(* IEC 61131-3 sources: smart-home/SmartHome/plc, 47 files *)

(* ---- Crosstable.gvl ---- *)
VAR_GLOBAL
	PLC_Iam_EP AT %QX0.4.0:BOOL;
	PLC_Iam_T1 AT %QX0.8.0:BOOL;
	PLC_Iam_T2 AT %QX0.12.0:BOOL;
	PLC_Iam_T3 AT %QX0.16.0:BOOL;
	PLC_Iam_T4 AT %QX0.20.0:BOOL;
	PLC_Iam_T5 AT %QX0.24.0:BOOL;
	PLC_Iam_T6 AT %QX0.28.0:BOOL;
	PLC_Iam_BA AT %QX0.32.0:BOOL;
	PLC_EP_exists AT %QX0.36.0:BOOL;
	PLC_Tn_count AT %QW0.40:UINT;	(* 0..6 *)
	PLC_BA_exists AT %QX0.44.0:BOOL;
	PLC_sunrise AT %QW0.48:UINT;	(* hh * 100 + mm *)
	PLC_sunset AT %QW0.52:UINT;	(* hh * 100 + mm *)
	PLC_day_brightness AT %QW0.56:UINT;
	PLC_night_brightness AT %QW0.60:UINT;
	PLC_screensaver AT %QW0.64:UINT;
	PLC_control_type AT %QW0.68:UINT;
	PLC_ConfigPassword AT %QD0.72:DINT;
	PLC_EP_enabled_wattmeters AT %QW0.80:UINT;	(* 0 .. 12 *)
	PLC_EP_enabled_relays AT %QW0.84:INT;	(* 0 .. 8 *)
	PLC_EP_overload_W AT %QW0.88:UINT;
	PLC_EP_max_assigned_W AT %QW0.92:UINT;
	PLC_EP_wattmeter_M_kWh_offset AT %QD0.96:DINT;	(* xxxxxxxxx.x kWh *)
	PLC_EP_wattmeter_M_e_kWh_offset AT %QD0.100:DINT;	(* xxxxxxxxx.x kWh *)
	PLC_EP_wattmeter_F_kWh_offset AT %QD0.104:DINT;	(* xxxxxxxxx.x kWh *)
	PLC_EP_wattmeter_F_e_kWh_offset AT %QD0.108:DINT;	(* xxxxxxxxx.x kWh *)
	PLC_EP_wattmeter01_kWh_offset AT %QD0.112:DINT;	(* xxxxxxxxx.x kWh *)
	PLC_EP_wattmeter02_kWh_offset AT %QD0.116:DINT;	(* xxxxxxxxx.x kWh *)
	PLC_EP_wattmeter03_kWh_offset AT %QD0.120:DINT;	(* xxxxxxxxx.x kWh *)
	PLC_EP_wattmeter04_kWh_offset AT %QD0.124:DINT;	(* xxxxxxxxx.x kWh *)
	PLC_EP_wattmeter05_kWh_offset AT %QD0.128:DINT;	(* xxxxxxxxx.x kWh *)
	PLC_EP_wattmeter06_kWh_offset AT %QD0.132:DINT;	(* xxxxxxxxx.x kWh *)
	PLC_EP_wattmeter07_kWh_offset AT %QD0.136:DINT;	(* xxxxxxxxx.x kWh *)
	PLC_EP_wattmeter08_kWh_offset AT %QD0.140:DINT;	(* xxxxxxxxx.x kWh *)
	PLC_EP_wattmeter09_kWh_offset AT %QD0.144:DINT;	(* xxxxxxxxx.x kWh *)
	PLC_EP_wattmeter10_kWh_offset AT %QD0.148:DINT;	(* xxxxxxxxx.x kWh *)
	PLC_T1_enabled_sensors AT %QW0.160:INT;
	PLC_T1_enabled_lamps AT %QW0.164:UINT;
	PLC_T1_max_request_W AT %QW0.168:UINT;
	PLC_T1_temperature_setpoint AT %QW0.172:INT;
	PLC_T1_humidity_setpoint AT %QW0.176:INT;
	PLC_T1_heating_status AT %QW0.180:INT;
	PLC_T1_temperature_setpoint_nt AT %QW0.184:INT;
	PLC_T1_humidity_setpoint_nt AT %QW0.188:INT;
	PLC_T1_daily_heating_s AT %QD0.192:UDINT;
	PLC_T1_monthly_heating_s AT %QD0.196:UDINT;
	PLC_T2_enabled_sensors AT %QW0.200:INT;
	PLC_T2_enabled_lamps AT %QW0.204:UINT;
	PLC_T2_max_request_W AT %QW0.208:UINT;
	PLC_T2_temperature_setpoint AT %QW0.212:INT;
	PLC_T2_humidity_setpoint AT %QW0.216:INT;
	PLC_T2_heating_status AT %QW0.220:INT;
	PLC_T2_temperature_setpoint_nt AT %QW0.224:INT;
	PLC_T2_humidity_setpoint_nt AT %QW0.228:INT;
	PLC_T2_daily_heating_s AT %QD0.232:UDINT;
	PLC_T2_monthly_heating_s AT %QD0.236:UDINT;
	PLC_T3_enabled_sensors AT %QW0.240:INT;
	PLC_T3_enabled_lamps AT %QW0.244:UINT;
	PLC_T3_max_request_W AT %QW0.248:UINT;
	PLC_T3_temperature_setpoint AT %QW0.252:INT;
	PLC_T3_humidity_setpoint AT %QW0.256:INT;
	PLC_T3_heating_status AT %QW0.260:INT;
	PLC_T3_temperature_setpoint_nt AT %QW0.264:INT;
	PLC_T3_humidity_setpoint_nt AT %QW0.268:INT;
	PLC_T3_daily_heating_s AT %QD0.272:UDINT;
	PLC_T3_monthly_heating_s AT %QD0.276:UDINT;
	PLC_T4_enabled_sensors AT %QW0.280:INT;
	PLC_T4_enabled_lamps AT %QW0.284:UINT;
	PLC_T4_max_request_W AT %QW0.288:UINT;
	PLC_T4_temperature_setpoint AT %QW0.292:INT;
	PLC_T4_humidity_setpoint AT %QW0.296:INT;
	PLC_T4_heating_status AT %QW0.300:INT;
	PLC_T4_temperature_setpoint_nt AT %QW0.304:INT;
	PLC_T4_humidity_setpoint_nt AT %QW0.308:INT;
	PLC_T4_daily_heating_s AT %QD0.312:UDINT;
	PLC_T4_monthly_heating_s AT %QD0.316:UDINT;
	PLC_T5_enabled_sensors AT %QW0.320:INT;
	PLC_T5_enabled_lamps AT %QW0.324:UINT;
	PLC_T5_max_request_W AT %QW0.328:UINT;
	PLC_T5_temperature_setpoint AT %QW0.332:INT;
	PLC_T5_humidity_setpoint AT %QW0.336:INT;
	PLC_T5_heating_status AT %QW0.340:INT;
	PLC_T5_temperature_setpoint_nt AT %QW0.344:INT;
	PLC_T5_humidity_setpoint_nt AT %QW0.348:INT;
	PLC_T5_daily_heating_s AT %QD0.352:UDINT;
	PLC_T5_monthly_heating_s AT %QD0.356:UDINT;
	PLC_T6_enabled_sensors AT %QW0.360:INT;
	PLC_T6_enabled_lamps AT %QW0.364:UINT;
	PLC_T6_max_request_W AT %QW0.368:UINT;
	PLC_T6_temperature_setpoint AT %QW0.372:INT;
	PLC_T6_humidity_setpoint AT %QW0.376:INT;
	PLC_T6_heating_status AT %QW0.380:INT;
	PLC_T6_temperature_setpoint_nt AT %QW0.384:INT;
	PLC_T6_humidity_setpoint_nt AT %QW0.388:INT;
	PLC_T6_daily_heating_s AT %QD0.392:UDINT;
	PLC_T6_monthly_heating_s AT %QD0.396:UDINT;
	PLC_BA_enabled_sensors AT %QW0.400:UINT;	(* 0, 8, 16, 24, 32 *)
	PLC_BA_daytime_bitmask AT %QD0.404:UDINT;
	PLC_BA_nighttime_bitmask AT %QD0.408:UDINT;
	PLC_BA_everything_bitmask AT %QD0.412:UDINT;
	PLC_BA_status AT %QW0.416:UINT;	(* ZERO, OFF, ARMED, ENABLED, RINGING, MUTED, TESTING *)
	PLC_BA_config_index AT %QW0.420:UINT;	(* 0 1 2 3 *)
	PLC_BA_password AT %QD0.424:DINT;
	Tsoglia_Resistenze AT %QW0.740:INT;	(* massima temperatura resistenze (50 .. 135 C) *)
	Tsoglia_Massetto AT %QW0.744:INT;	(* massima temperatura massetto (20 .. 30 C) *)
	Tsoglia_Ventola AT %QW0.748:INT;	(* minima temperatura ventole (50 .. 125 C) *)
	Vbase_Ventola AT %QW0.752:UINT;	(* valore base comando ventola (1.00V ..) *)
	TimerValue_1 AT %QD0.760:DINT;
	TimerValue_2 AT %QD0.764:DINT;
	PLC_RELOAD_CONF AT %QX0.772.0:BOOL;
	PLC_BA_just_started AT %QX0.776.0:BOOL;	(* just after init *)
	PLC_view_passwords AT %QX0.780.0:BOOL;
	PLC_buzzer_timer_1 AT %QX0.784.0:BOOL;
	PLC_buzzer_timer_2 AT %QX0.788.0:BOOL;
	PLC_buzzer_alarm AT %QX0.792.0:BOOL;
	PLC_buzzer_blackout_or_overload AT %QX0.796.0:BOOL;
	PLC_BA_ringing_flag AT %QX0.800.0:BOOL;
	PLC_BA_blackout_digin AT %QX0.804.0:BOOL;	(* Blackout detected flag *)
	PLC_EP_blackout_flag AT %QX0.808.0:BOOL;	(* Blackout detected flag *)
	PLC_EP_overload_flag AT %QX0.812.0:BOOL;	(* Overload detected flag *)
	PLC_EP_isOK AT %QX0.816.0:BOOL;
	PLC_T1_isOK AT %QX0.820.0:BOOL;
	PLC_T2_isOK AT %QX0.824.0:BOOL;
	PLC_T3_isOK AT %QX0.828.0:BOOL;
	PLC_T4_isOK AT %QX0.832.0:BOOL;
	PLC_T5_isOK AT %QX0.836.0:BOOL;
	PLC_T6_isOK AT %QX0.840.0:BOOL;
	PLC_BA_isOK AT %QX0.868.0:BOOL;
	PLC_BA_AlarmRinging AT %IX0.872.0:BOOL;	(* BA Alarm is ringing *)
	PLC_BA_BlackoutDetected AT %IX0.876.0:BOOL;	(* BA Blackout detected *)
	PLC_EP_BlackoutDetected AT %IX0.880.0:BOOL;	(* EP Blackout detected *)
	PLC_EP_OverloadDetected AT %IX0.884.0:BOOL;	(* EP Overload detected *)
	PLC_nighttime AT %QX0.888.0:BOOL;
	PLC_Tn_heating AT %QX0.892.0:BOOL;	(* al least one Tn is heating *)
	PLC_time_bis AT %QD0.912:REAL;	(* PLC_time + PLC_timeOffset *)
	PLC_timeMin_bis AT %QD0.916:REAL;	(* PLC_timeMin + PLC_timeOffset *)
	PLC_timeMax_bis AT %QD0.920:REAL;	(* PLC_timeMax + PLC_timeOffset *)
	PLC_timeOffset AT %QD0.924:REAL;	(* Graph display window *)
	TCP_EP_heartbeat AT %IW0.4000:UINT;	(* TCPS_STATUS NODE_09_STATUS *)
	TCP_EP_enabled_wattmeters AT %IW0.4004:UINT;	(* 0 .. 12 *)
	TCP_EP_wattmeters_ok AT %IW0.4008:UINT;	(* bit mask (node status) *)
	TCP_EP_wattmeter_M_W AT %IW0.4012:INT;	(* +/- xxxx W *)
	TCP_EP_wattmeter_M_var AT %IW0.4016:INT;	(* +/- xxxx var *)
	TCP_EP_wattmeter_M_VA AT %IW0.4020:INT;	(* +/- xxxx VA *)
	TCP_EP_wattmeter_M_pf AT %IW0.4024:INT;	(* +/- x.xxx *)
	TCP_EP_wattmeter_M_Hz AT %IW0.4028:INT;	(* xxx.xx Hz *)
	TCP_EP_wattmeter_M_V AT %IW0.4032:INT;	(* xxx.xx V *)
	TCP_EP_wattmeter_M_A AT %IW0.4036:INT;	(* xx.xxx A *)
	TCP_EP_wattmeter_M_kWh AT %ID0.4040:DINT;	(* xxxxxxxxx.x +kWh *)
	TCP_EP_wattmeter_M_e_kWh AT %ID0.4044:DINT;	(* xxxxxxxxx.x -kWh *)
	TCP_EP_wattmeter_F_W AT %IW0.4048:INT;	(* +/- xxxx W *)
	TCP_EP_wattmeter_F_var AT %IW0.4052:INT;	(* +/- xxxx var *)
	TCP_EP_wattmeter_F_VA AT %IW0.4056:INT;	(* +/- xxxx VA *)
	TCP_EP_wattmeter_F_pf AT %IW0.4060:INT;	(* +/- x.xxx *)
	TCP_EP_wattmeter_F_Hz AT %IW0.4064:INT;	(* xxx.xx Hz *)
	TCP_EP_wattmeter_F_V AT %IW0.4068:INT;	(* xxx.xx V *)
	TCP_EP_wattmeter_F_A AT %IW0.4072:INT;	(* xx.xxx A *)
	TCP_EP_wattmeter_F_kWh AT %ID0.4076:DINT;	(* xxxxxxxxx.x +kWh *)
	TCP_EP_wattmeter_F_e_kWh AT %ID0.4080:DINT;	(* xxxxxxxxx.x -kWh *)
	TCP_EP_wattmeter01_W AT %IW0.4084:INT;	(* +/- xxxx W *)
	TCP_EP_wattmeter01_var AT %IW0.4088:INT;	(* +/- xxxx var *)
	TCP_EP_wattmeter01_VA AT %IW0.4092:INT;	(* +/- xxxx VA *)
	TCP_EP_wattmeter01_kWh AT %ID0.4096:DINT;	(* xxxxxxxxx.x +kWh *)
	TCP_EP_wattmeter02_W AT %IW0.4100:INT;	(* +/- xxxx W *)
	TCP_EP_wattmeter02_var AT %IW0.4104:INT;	(* +/- xxxx var *)
	TCP_EP_wattmeter02_VA AT %IW0.4108:INT;	(* +/- xxxx VA *)
	TCP_EP_wattmeter02_kWh AT %ID0.4112:DINT;	(* xxxxxxxxx.x +kWh *)
	TCP_EP_wattmeter03_W AT %IW0.4116:INT;	(* +/- xxxx W *)
	TCP_EP_wattmeter03_var AT %IW0.4120:INT;	(* +/- xxxx var *)
	TCP_EP_wattmeter03_VA AT %IW0.4124:INT;	(* +/- xxxx VA *)
	TCP_EP_wattmeter03_kWh AT %ID0.4128:DINT;	(* xxxxxxxxx.x +kWh *)
	TCP_EP_wattmeter04_W AT %IW0.4132:INT;	(* +/- xxxx W *)
	TCP_EP_wattmeter04_var AT %IW0.4136:INT;	(* +/- xxxx var *)
	TCP_EP_wattmeter04_VA AT %IW0.4140:INT;	(* +/- xxxx VA *)
	TCP_EP_wattmeter04_kWh AT %ID0.4144:DINT;	(* xxxxxxxxx.x +kWh *)
	TCP_EP_wattmeter05_W AT %IW0.4148:INT;	(* +/- xxxx W *)
	TCP_EP_wattmeter05_var AT %IW0.4152:INT;	(* +/- xxxx var *)
	TCP_EP_wattmeter05_VA AT %IW0.4156:INT;	(* +/- xxxx VA *)
	TCP_EP_wattmeter05_kWh AT %ID0.4160:DINT;	(* xxxxxxxxx.x +kWh *)
	TCP_EP_wattmeter06_W AT %IW0.4164:INT;	(* +/- xxxx W *)
	TCP_EP_wattmeter06_var AT %IW0.4168:INT;	(* +/- xxxx var *)
	TCP_EP_wattmeter06_VA AT %IW0.4172:INT;	(* +/- xxxx VA *)
	TCP_EP_wattmeter06_kWh AT %ID0.4176:DINT;	(* xxxxxxxxx.x +kWh *)
	TCP_EP_wattmeter07_W AT %IW0.4180:INT;	(* +/- xxxx W *)
	TCP_EP_wattmeter07_var AT %IW0.4184:INT;	(* +/- xxxx var *)
	TCP_EP_wattmeter07_VA AT %IW0.4188:INT;	(* +/- xxxx VA *)
	TCP_EP_wattmeter07_kWh AT %ID0.4192:DINT;	(* xxxxxxxxx.x +kWh *)
	TCP_EP_wattmeter08_W AT %IW0.4196:INT;	(* +/- xxxx W *)
	TCP_EP_wattmeter08_var AT %IW0.4200:INT;	(* +/- xxxx var *)
	TCP_EP_wattmeter08_VA AT %IW0.4204:INT;	(* +/- xxxx VA *)
	TCP_EP_wattmeter08_kWh AT %ID0.4208:DINT;	(* xxxxxxxxx.x +kWh *)
	TCP_EP_wattmeter09_W AT %IW0.4212:INT;	(* +/- xxxx W *)
	TCP_EP_wattmeter09_var AT %IW0.4216:INT;	(* +/- xxxx var *)
	TCP_EP_wattmeter09_VA AT %IW0.4220:INT;	(* +/- xxxx VA *)
	TCP_EP_wattmeter09_kWh AT %ID0.4224:DINT;	(* xxxxxxxxx.x +kWh *)
	TCP_EP_wattmeter10_W AT %IW0.4228:INT;	(* +/- xxxx W *)
	TCP_EP_wattmeter10_var AT %IW0.4232:INT;	(* +/- xxxx var *)
	TCP_EP_wattmeter10_VA AT %IW0.4236:INT;	(* +/- xxxx VA *)
	TCP_EP_wattmeter10_kWh AT %ID0.4240:DINT;	(* xxxxxxxxx.x +kWh *)
	TCP_EP_BlackoutDetected AT %IX0.4244.0:BOOL;
	TCP_EP_OverloadDetected AT %IX0.4248.0:BOOL;
	TCP_EP_enabled_relays AT %IW0.4252:INT;	(* 0 .. 8 *)
	TCP_EP_relay_A AT %QX0.4256.0:BOOL;
	TCP_EP_relay_B AT %QX0.4260.0:BOOL;
	TCP_EP_relay_C AT %QX0.4264.0:BOOL;
	TCP_EP_relay_D AT %QX0.4268.0:BOOL;
	TCP_EP_relay_E AT %QX0.4272.0:BOOL;
	TCP_EP_relay_F AT %QX0.4276.0:BOOL;
	TCP_EP_relay_G AT %QX0.4280.0:BOOL;
	TCP_EP_relay_H AT %QX0.4284.0:BOOL;
	TCP_EP_overload_W AT %IW0.4288:UINT;
	TCP_EP_max_assigned_W AT %IW0.4292:UINT;
	TCP_EP_tic_in_tac AT %IW0.4296:UINT;
	TCP_EP_requested_W AT %IW0.4300:UINT;
	TCP_EP_T1_assigned_W AT %IW0.4304:UINT;
	TCP_EP_T2_assigned_W AT %IW0.4308:UINT;
	TCP_EP_T3_assigned_W AT %IW0.4312:UINT;
	TCP_EP_T4_assigned_W AT %IW0.4316:UINT;
	TCP_EP_T5_assigned_W AT %IW0.4320:UINT;
	TCP_EP_T6_assigned_W AT %IW0.4324:UINT;
	TCP_EP_assigned_W AT %IW0.4328:UINT;
	TCP_EP_control_type AT %IW0.4332:UINT;
	TCP_T1_heartbeat AT %IW0.4400:UINT;	(* TCP1_STATUS NODE_02_STATUS *)
	TCP_T1_enabled_sensors AT %IW0.4404:INT;
	TCP_T1_temperature AT %IW0.4408:INT;
	TCP_T1_temperature_bis AT %IW0.4412:INT;
	TCP_T1_temperature_ext AT %IW0.4416:INT;
	TCP_T1_humidity AT %IW0.4420:INT;
	TCP_T1_humidity_bis AT %IW0.4424:INT;
	TCP_T1_humidity_ext AT %IW0.4428:INT;
	TCP_T1_temperature_setpoint AT %QW0.4432:INT;
	TCP_T1_humidity_setpoint AT %QW0.4436:INT;
	TCP_T1_enabled_lamps AT %IW0.4440:UINT;
	TCP_T1_lamp_1 AT %QX0.4444.0:BOOL;
	TCP_T1_lamp_2 AT %QX0.4448.0:BOOL;
	TCP_T1_lamp_3 AT %QX0.4452.0:BOOL;
	TCP_T1_lamp_4 AT %QX0.4456.0:BOOL;
	TCP_T1_lamp_5 AT %QX0.4460.0:BOOL;
	TCP_T1_max_request_W AT %IW0.4464:UINT;
	TCP_T1_heating AT %IX0.4468.0:BOOL;
	TCP_T1_nighttime AT %IX0.4472.0:BOOL;
	TCP_T1_heating_status AT %QW0.4476:INT;
	TCP_T1_heating_timer AT %QW0.4480:INT;	(* seconds (max 9 h) *)
	TCP_T1_sunrise AT %QW0.4484:UINT;	(* hh * 100 + mm *)
	TCP_T1_sunset AT %QW0.4488:UINT;	(* hh * 100 + mm *)
	TCP_T1_temperature_setpoint_nt AT %QW0.4492:INT;
	TCP_T1_humidity_setpoint_nt AT %QW0.4496:INT;
	TCP_T1_lamp_feedback_1 AT %IX0.4500.0:BOOL;
	TCP_T1_lamp_feedback_2 AT %IX0.4504.0:BOOL;
	TCP_T1_lamp_feedback_3 AT %IX0.4508.0:BOOL;
	TCP_T1_lamp_feedback_4 AT %IX0.4512.0:BOOL;
	TCP_T1_lamp_feedback_5 AT %IX0.4516.0:BOOL;
	TCP_T1_requested_W AT %IW0.4520:UINT;
	TCP_T1_control_type AT %IW0.4524:UINT;
	TCP_T1_daily_heating_s AT %ID0.4528:UDINT;
	TCP_T1_monthly_heating_s AT %ID0.4532:UDINT;
	TCP_T2_heartbeat AT %IW0.4600:UINT;	(* TCP2_STATUS NODE_03_STATUS *)
	TCP_T2_enabled_sensors AT %IW0.4604:INT;
	TCP_T2_temperature AT %IW0.4608:INT;
	TCP_T2_temperature_bis AT %IW0.4612:INT;
	TCP_T2_temperature_ext AT %IW0.4616:INT;
	TCP_T2_humidity AT %IW0.4620:INT;
	TCP_T2_humidity_bis AT %IW0.4624:INT;
	TCP_T2_humidity_ext AT %IW0.4628:INT;
	TCP_T2_temperature_setpoint AT %QW0.4632:INT;
	TCP_T2_humidity_setpoint AT %QW0.4636:INT;
	TCP_T2_enabled_lamps AT %IW0.4640:UINT;
	TCP_T2_lamp_1 AT %QX0.4644.0:BOOL;
	TCP_T2_lamp_2 AT %QX0.4648.0:BOOL;
	TCP_T2_lamp_3 AT %QX0.4652.0:BOOL;
	TCP_T2_lamp_4 AT %QX0.4656.0:BOOL;
	TCP_T2_lamp_5 AT %QX0.4660.0:BOOL;
	TCP_T2_max_request_W AT %IW0.4664:UINT;
	TCP_T2_heating AT %IX0.4668.0:BOOL;
	TCP_T2_nighttime AT %IX0.4672.0:BOOL;
	TCP_T2_heating_status AT %QW0.4676:INT;
	TCP_T2_heating_timer AT %QW0.4680:INT;	(* seconds (max 9 h) *)
	TCP_T2_sunrise AT %QW0.4684:UINT;	(* hh * 100 + mm *)
	TCP_T2_sunset AT %QW0.4688:UINT;	(* hh * 100 + mm *)
	TCP_T2_temperature_setpoint_nt AT %QW0.4692:INT;
	TCP_T2_humidity_setpoint_nt AT %QW0.4696:INT;
	TCP_T2_lamp_feedback_1 AT %IX0.4700.0:BOOL;
	TCP_T2_lamp_feedback_2 AT %IX0.4704.0:BOOL;
	TCP_T2_lamp_feedback_3 AT %IX0.4708.0:BOOL;
	TCP_T2_lamp_feedback_4 AT %IX0.4712.0:BOOL;
	TCP_T2_lamp_feedback_5 AT %IX0.4716.0:BOOL;
	TCP_T2_requested_W AT %IW0.4720:UINT;
	TCP_T2_control_type AT %IW0.4724:UINT;
	TCP_T2_daily_heating_s AT %ID0.4728:UDINT;
	TCP_T2_monthly_heating_s AT %ID0.4732:UDINT;
	TCP_T3_heartbeat AT %IW0.4800:UINT;	(* TCP3_STATUS NODE_04_STATUS *)
	TCP_T3_enabled_sensors AT %IW0.4804:INT;
	TCP_T3_temperature AT %IW0.4808:INT;
	TCP_T3_temperature_bis AT %IW0.4812:INT;
	TCP_T3_temperature_ext AT %IW0.4816:INT;
	TCP_T3_humidity AT %IW0.4820:INT;
	TCP_T3_humidity_bis AT %IW0.4824:INT;
	TCP_T3_humidity_ext AT %IW0.4828:INT;
	TCP_T3_temperature_setpoint AT %QW0.4832:INT;
	TCP_T3_humidity_setpoint AT %QW0.4836:INT;
	TCP_T3_enabled_lamps AT %IW0.4840:UINT;
	TCP_T3_lamp_1 AT %QX0.4844.0:BOOL;
	TCP_T3_lamp_2 AT %QX0.4848.0:BOOL;
	TCP_T3_lamp_3 AT %QX0.4852.0:BOOL;
	TCP_T3_lamp_4 AT %QX0.4856.0:BOOL;
	TCP_T3_lamp_5 AT %QX0.4860.0:BOOL;
	TCP_T3_max_request_W AT %IW0.4864:UINT;
	TCP_T3_heating AT %IX0.4868.0:BOOL;
	TCP_T3_nighttime AT %IX0.4872.0:BOOL;
	TCP_T3_heating_status AT %QW0.4876:INT;
	TCP_T3_heating_timer AT %QW0.4880:INT;	(* seconds (max 9 h) *)
	TCP_T3_sunrise AT %QW0.4884:UINT;	(* hh * 100 + mm *)
	TCP_T3_sunset AT %QW0.4888:UINT;	(* hh * 100 + mm *)
	TCP_T3_temperature_setpoint_nt AT %QW0.4892:INT;
	TCP_T3_humidity_setpoint_nt AT %QW0.4896:INT;
	TCP_T3_lamp_feedback_1 AT %IX0.4900.0:BOOL;
	TCP_T3_lamp_feedback_2 AT %IX0.4904.0:BOOL;
	TCP_T3_lamp_feedback_3 AT %IX0.4908.0:BOOL;
	TCP_T3_lamp_feedback_4 AT %IX0.4912.0:BOOL;
	TCP_T3_lamp_feedback_5 AT %IX0.4916.0:BOOL;
	TCP_T3_requested_W AT %IW0.4920:UINT;
	TCP_T3_control_type AT %IW0.4924:UINT;
	TCP_T3_daily_heating_s AT %ID0.4928:UDINT;
	TCP_T3_monthly_heating_s AT %ID0.4932:UDINT;
	TCP_T4_heartbeat AT %IW0.5000:UINT;	(* TCP4_STATUS NODE_05_STATUS *)
	TCP_T4_enabled_sensors AT %IW0.5004:INT;
	TCP_T4_temperature AT %IW0.5008:INT;
	TCP_T4_temperature_bis AT %IW0.5012:INT;
	TCP_T4_temperature_ext AT %IW0.5016:INT;
	TCP_T4_humidity AT %IW0.5020:INT;
	TCP_T4_humidity_bis AT %IW0.5024:INT;
	TCP_T4_humidity_ext AT %IW0.5028:INT;
	TCP_T4_temperature_setpoint AT %QW0.5032:INT;
	TCP_T4_humidity_setpoint AT %QW0.5036:INT;
	TCP_T4_enabled_lamps AT %IW0.5040:UINT;
	TCP_T4_lamp_1 AT %QX0.5044.0:BOOL;
	TCP_T4_lamp_2 AT %QX0.5048.0:BOOL;
	TCP_T4_lamp_3 AT %QX0.5052.0:BOOL;
	TCP_T4_lamp_4 AT %QX0.5056.0:BOOL;
	TCP_T4_lamp_5 AT %QX0.5060.0:BOOL;
	TCP_T4_max_request_W AT %IW0.5064:UINT;
	TCP_T4_heating AT %IX0.5068.0:BOOL;
	TCP_T4_nighttime AT %IX0.5072.0:BOOL;
	TCP_T4_heating_status AT %QW0.5076:INT;
	TCP_T4_heating_timer AT %QW0.5080:INT;	(* seconds (max 9 h) *)
	TCP_T4_sunrise AT %QW0.5084:UINT;	(* hh * 100 + mm *)
	TCP_T4_sunset AT %QW0.5088:UINT;	(* hh * 100 + mm *)
	TCP_T4_temperature_setpoint_nt AT %QW0.5092:INT;
	TCP_T4_humidity_setpoint_nt AT %QW0.5096:INT;
	TCP_T4_lamp_feedback_1 AT %IX0.5100.0:BOOL;
	TCP_T4_lamp_feedback_2 AT %IX0.5104.0:BOOL;
	TCP_T4_lamp_feedback_3 AT %IX0.5108.0:BOOL;
	TCP_T4_lamp_feedback_4 AT %IX0.5112.0:BOOL;
	TCP_T4_lamp_feedback_5 AT %IX0.5116.0:BOOL;
	TCP_T4_requested_W AT %IW0.5120:UINT;
	TCP_T4_control_type AT %IW0.5124:UINT;
	TCP_T4_daily_heating_s AT %ID0.5128:UDINT;
	TCP_T4_monthly_heating_s AT %ID0.5132:UDINT;
	TCP_T5_heartbeat AT %IW0.5200:UINT;	(* TCP5_STATUS NODE_06_STATUS *)
	TCP_T5_enabled_sensors AT %IW0.5204:INT;
	TCP_T5_temperature AT %IW0.5208:INT;
	TCP_T5_temperature_bis AT %IW0.5212:INT;
	TCP_T5_temperature_ext AT %IW0.5216:INT;
	TCP_T5_humidity AT %IW0.5220:INT;
	TCP_T5_humidity_bis AT %IW0.5224:INT;
	TCP_T5_humidity_ext AT %IW0.5228:INT;
	TCP_T5_temperature_setpoint AT %QW0.5232:INT;
	TCP_T5_humidity_setpoint AT %QW0.5236:INT;
	TCP_T5_enabled_lamps AT %IW0.5240:UINT;
	TCP_T5_lamp_1 AT %QX0.5244.0:BOOL;
	TCP_T5_lamp_2 AT %QX0.5248.0:BOOL;
	TCP_T5_lamp_3 AT %QX0.5252.0:BOOL;
	TCP_T5_lamp_4 AT %QX0.5256.0:BOOL;
	TCP_T5_lamp_5 AT %QX0.5260.0:BOOL;
	TCP_T5_max_request_W AT %IW0.5264:UINT;
	TCP_T5_heating AT %IX0.5268.0:BOOL;
	TCP_T5_nighttime AT %IX0.5272.0:BOOL;
	TCP_T5_heating_status AT %QW0.5276:INT;
	TCP_T5_heating_timer AT %QW0.5280:INT;	(* seconds (max 9 h) *)
	TCP_T5_sunrise AT %QW0.5284:UINT;	(* hh * 100 + mm *)
	TCP_T5_sunset AT %QW0.5288:UINT;	(* hh * 100 + mm *)
	TCP_T5_temperature_setpoint_nt AT %QW0.5292:INT;
	TCP_T5_humidity_setpoint_nt AT %QW0.5296:INT;
	TCP_T5_lamp_feedback_1 AT %IX0.5300.0:BOOL;
	TCP_T5_lamp_feedback_2 AT %IX0.5304.0:BOOL;
	TCP_T5_lamp_feedback_3 AT %IX0.5308.0:BOOL;
	TCP_T5_lamp_feedback_4 AT %IX0.5312.0:BOOL;
	TCP_T5_lamp_feedback_5 AT %IX0.5316.0:BOOL;
	TCP_T5_requested_W AT %IW0.5320:UINT;
	TCP_T5_control_type AT %IW0.5324:UINT;
	TCP_T5_daily_heating_s AT %ID0.5328:UDINT;
	TCP_T5_monthly_heating_s AT %ID0.5332:UDINT;
	TCP_T6_heartbeat AT %IW0.5400:UINT;	(* TCP6_STATUS NODE_07_STATUS *)
	TCP_T6_enabled_sensors AT %IW0.5404:INT;
	TCP_T6_temperature AT %IW0.5408:INT;
	TCP_T6_temperature_bis AT %IW0.5412:INT;
	TCP_T6_temperature_ext AT %IW0.5416:INT;
	TCP_T6_humidity AT %IW0.5420:INT;
	TCP_T6_humidity_bis AT %IW0.5424:INT;
	TCP_T6_humidity_ext AT %IW0.5428:INT;
	TCP_T6_temperature_setpoint AT %QW0.5432:INT;
	TCP_T6_humidity_setpoint AT %QW0.5436:INT;
	TCP_T6_enabled_lamps AT %IW0.5440:UINT;
	TCP_T6_lamp_1 AT %QX0.5444.0:BOOL;
	TCP_T6_lamp_2 AT %QX0.5448.0:BOOL;
	TCP_T6_lamp_3 AT %QX0.5452.0:BOOL;
	TCP_T6_lamp_4 AT %QX0.5456.0:BOOL;
	TCP_T6_lamp_5 AT %QX0.5460.0:BOOL;
	TCP_T6_max_request_W AT %IW0.5464:UINT;
	TCP_T6_heating AT %IX0.5468.0:BOOL;
	TCP_T6_nighttime AT %IX0.5472.0:BOOL;
	TCP_T6_heating_status AT %QW0.5476:INT;
	TCP_T6_heating_timer AT %QW0.5480:INT;	(* seconds (max 9 h) *)
	TCP_T6_sunrise AT %QW0.5484:UINT;	(* hh * 100 + mm *)
	TCP_T6_sunset AT %QW0.5488:UINT;	(* hh * 100 + mm *)
	TCP_T6_temperature_setpoint_nt AT %QW0.5492:INT;
	TCP_T6_humidity_setpoint_nt AT %QW0.5496:INT;
	TCP_T6_lamp_feedback_1 AT %IX0.5500.0:BOOL;
	TCP_T6_lamp_feedback_2 AT %IX0.5504.0:BOOL;
	TCP_T6_lamp_feedback_3 AT %IX0.5508.0:BOOL;
	TCP_T6_lamp_feedback_4 AT %IX0.5512.0:BOOL;
	TCP_T6_lamp_feedback_5 AT %IX0.5516.0:BOOL;
	TCP_T6_requested_W AT %IW0.5520:UINT;
	TCP_T6_control_type AT %IW0.5524:UINT;
	TCP_T6_daily_heating_s AT %ID0.5528:UDINT;
	TCP_T6_monthly_heating_s AT %ID0.5532:UDINT;
	TCP_BA_heartbeat AT %IW0.6800:UINT;	(* TCP7_STATUS NODE_08_STATUS *)
	TCP_BA_enabled_sensors AT %IW0.6804:UINT;	(* 0, 8, 16, 24, 32 *)
	TCP_BA_status AT %IW0.6808:UINT;	(* ZERO, OFF, ARMED, ENABLED, RINGING, MUTED, TESTING *)
	TCP_BA_config_index AT %IW0.6812:UINT;	(* 0 1 2 3 *)
	TCP_BA_config_mask AT %ID0.6816:UDINT;	(* bit mask *)
	TCP_BA_led_green AT %IX0.6820.0:BOOL;	(* ARMED(blinking), ENABLED, RINGING, MUTED *)
	TCP_BA_led_red AT %IX0.6824.0:BOOL;	(* ARMED(if NG), RINGING(blinking), MUTED *)
	TCP_BA_led_yellow1 AT %IX0.6828.0:BOOL;	(* NIGHTIME, EVERYTHING *)
	TCP_BA_led_yellow2 AT %IX0.6832.0:BOOL;	(* DAYTIME, EVERYTHING *)
	TCP_BA_siren AT %IX0.6836.0:BOOL;	(* HPA *)
	TCP_BA_relay_A AT %IX0.6840.0:BOOL;
	TCP_BA_relay_B AT %IX0.6844.0:BOOL;
	TCP_BA_relay_C AT %IX0.6848.0:BOOL;
	TCP_BA_input_9 AT %IX0.6852.0:BOOL;
	TCP_BA_input_10 AT %IX0.6856.0:BOOL;
	TCP_BA_input_11 AT %IX0.6860.0:BOOL;
	TCP_BA_input_12 AT %IX0.6864.0:BOOL;
	TCP_BA_BlackoutDetected AT %IX0.6868.0:BOOL;
	TCP_BA_command AT %QD0.6872:UDINT;	(* NONE, ARM, NOTHING, DAYTIME, NIGHTIME, EVERYTHING, ENABLE, DISABLE, ACK, TEST *)
	TCP_BA_OK_1 AT %IW0.6876:UINT;
	TCP_BA_OK_2 AT %IW0.6880:UINT;
	TCP_BA_OK_3 AT %IW0.6884:UINT;
	TCP_BA_OK_4 AT %IW0.6888:UINT;
	TCP_BA_OK_5 AT %IW0.6892:UINT;
	TCP_BA_OK_6 AT %IW0.6896:UINT;
	TCP_BA_OK_7 AT %IW0.6900:UINT;
	TCP_BA_OK_8 AT %IW0.6904:UINT;
	TCP_BA_OK_9 AT %IW0.6908:UINT;
	TCP_BA_OK_10 AT %IW0.6912:UINT;
	TCP_BA_OK_11 AT %IW0.6916:UINT;
	TCP_BA_OK_12 AT %IW0.6920:UINT;
	TCP_BA_OK_13 AT %IW0.6924:UINT;
	TCP_BA_OK_14 AT %IW0.6928:UINT;
	TCP_BA_OK_15 AT %IW0.6932:UINT;
	TCP_BA_OK_16 AT %IW0.6936:UINT;
	TCP_BA_OK_17 AT %IW0.6940:UINT;
	TCP_BA_OK_18 AT %IW0.6944:UINT;
	TCP_BA_OK_19 AT %IW0.6948:UINT;
	TCP_BA_OK_20 AT %IW0.6952:UINT;
	TCP_BA_OK_21 AT %IW0.6956:UINT;
	TCP_BA_OK_22 AT %IW0.6960:UINT;
	TCP_BA_OK_23 AT %IW0.6964:UINT;
	TCP_BA_OK_24 AT %IW0.6968:UINT;
	TCP_BA_OK_25 AT %IW0.6972:UINT;
	TCP_BA_OK_26 AT %IW0.6976:UINT;
	TCP_BA_OK_27 AT %IW0.6980:UINT;
	TCP_BA_OK_28 AT %IW0.6984:UINT;
	TCP_BA_OK_29 AT %IW0.6988:UINT;
	TCP_BA_OK_30 AT %IW0.6992:UINT;
	TCP_BA_OK_31 AT %IW0.6996:UINT;
	TCP_BA_OK_32 AT %IW0.7000:UINT;
	TCP_BA_control_type AT %IW0.7004:UINT;
	SRV_EP_heartbeat AT %QW0.8000:UINT;	(* TCPS_STATUS NODE_09_STATUS *)
	SRV_EP_enabled_wattmeters AT %QW0.8004:UINT;	(* 0 .. 12 *)
	SRV_EP_wattmeters_ok AT %QW0.8008:UINT;	(* bit mask (node status) *)
	SRV_EP_wattmeter_M_W AT %QW0.8012:INT;	(* +/- xxxx W *)
	SRV_EP_wattmeter_M_var AT %QW0.8016:INT;	(* +/- xxxx var *)
	SRV_EP_wattmeter_M_VA AT %QW0.8020:INT;	(* +/- xxxx VA *)
	SRV_EP_wattmeter_M_pf AT %QW0.8024:INT;	(* +/- x.xxx *)
	SRV_EP_wattmeter_M_Hz AT %QW0.8028:INT;	(* xxx.xx Hz *)
	SRV_EP_wattmeter_M_V AT %QW0.8032:INT;	(* xxx.xx V *)
	SRV_EP_wattmeter_M_A AT %QW0.8036:INT;	(* xx.xxx A *)
	SRV_EP_wattmeter_M_kWh AT %QD0.8040:DINT;	(* xxxxxxxxx.x +kWh *)
	SRV_EP_wattmeter_M_e_kWh AT %QD0.8044:DINT;	(* xxxxxxxxx.x -kWh *)
	SRV_EP_wattmeter_F_W AT %QW0.8048:INT;	(* +/- xxxx W *)
	SRV_EP_wattmeter_F_var AT %QW0.8052:INT;	(* +/- xxxx var *)
	SRV_EP_wattmeter_F_VA AT %QW0.8056:INT;	(* +/- xxxx VA *)
	SRV_EP_wattmeter_F_pf AT %QW0.8060:INT;	(* +/- x.xxx *)
	SRV_EP_wattmeter_F_Hz AT %QW0.8064:INT;	(* xxx.xx Hz *)
	SRV_EP_wattmeter_F_V AT %QW0.8068:INT;	(* xxx.xx V *)
	SRV_EP_wattmeter_F_A AT %QW0.8072:INT;	(* xx.xxx A *)
	SRV_EP_wattmeter_F_kWh AT %QD0.8076:DINT;	(* xxxxxxxxx.x +kWh *)
	SRV_EP_wattmeter_F_e_kWh AT %QD0.8080:DINT;	(* xxxxxxxxx.x -kWh *)
	SRV_EP_wattmeter01_W AT %QW0.8084:INT;	(* +/- xxxx W *)
	SRV_EP_wattmeter01_var AT %QW0.8088:INT;	(* +/- xxxx var *)
	SRV_EP_wattmeter01_VA AT %QW0.8092:INT;	(* +/- xxxx VA *)
	SRV_EP_wattmeter01_kWh AT %QD0.8096:DINT;	(* xxxxxxxxx.x +kWh *)
	SRV_EP_wattmeter02_W AT %QW0.8100:INT;	(* +/- xxxx W *)
	SRV_EP_wattmeter02_var AT %QW0.8104:INT;	(* +/- xxxx var *)
	SRV_EP_wattmeter02_VA AT %QW0.8108:INT;	(* +/- xxxx VA *)
	SRV_EP_wattmeter02_kWh AT %QD0.8112:DINT;	(* xxxxxxxxx.x +kWh *)
	SRV_EP_wattmeter03_W AT %QW0.8116:INT;	(* +/- xxxx W *)
	SRV_EP_wattmeter03_var AT %QW0.8120:INT;	(* +/- xxxx var *)
	SRV_EP_wattmeter03_VA AT %QW0.8124:INT;	(* +/- xxxx VA *)
	SRV_EP_wattmeter03_kWh AT %QD0.8128:DINT;	(* xxxxxxxxx.x +kWh *)
	SRV_EP_wattmeter04_W AT %QW0.8132:INT;	(* +/- xxxx W *)
	SRV_EP_wattmeter04_var AT %QW0.8136:INT;	(* +/- xxxx var *)
	SRV_EP_wattmeter04_VA AT %QW0.8140:INT;	(* +/- xxxx VA *)
	SRV_EP_wattmeter04_kWh AT %QD0.8144:DINT;	(* xxxxxxxxx.x +kWh *)
	SRV_EP_wattmeter05_W AT %QW0.8148:INT;	(* +/- xxxx W *)
	SRV_EP_wattmeter05_var AT %QW0.8152:INT;	(* +/- xxxx var *)
	SRV_EP_wattmeter05_VA AT %QW0.8156:INT;	(* +/- xxxx VA *)
	SRV_EP_wattmeter05_kWh AT %QD0.8160:DINT;	(* xxxxxxxxx.x +kWh *)
	SRV_EP_wattmeter06_W AT %QW0.8164:INT;	(* +/- xxxx W *)
	SRV_EP_wattmeter06_var AT %QW0.8168:INT;	(* +/- xxxx var *)
	SRV_EP_wattmeter06_VA AT %QW0.8172:INT;	(* +/- xxxx VA *)
	SRV_EP_wattmeter06_kWh AT %QD0.8176:DINT;	(* xxxxxxxxx.x +kWh *)
	SRV_EP_wattmeter07_W AT %QW0.8180:INT;	(* +/- xxxx W *)
	SRV_EP_wattmeter07_var AT %QW0.8184:INT;	(* +/- xxxx var *)
	SRV_EP_wattmeter07_VA AT %QW0.8188:INT;	(* +/- xxxx VA *)
	SRV_EP_wattmeter07_kWh AT %QD0.8192:DINT;	(* xxxxxxxxx.x +kWh *)
	SRV_EP_wattmeter08_W AT %QW0.8196:INT;	(* +/- xxxx W *)
	SRV_EP_wattmeter08_var AT %QW0.8200:INT;	(* +/- xxxx var *)
	SRV_EP_wattmeter08_VA AT %QW0.8204:INT;	(* +/- xxxx VA *)
	SRV_EP_wattmeter08_kWh AT %QD0.8208:DINT;	(* xxxxxxxxx.x +kWh *)
	SRV_EP_wattmeter09_W AT %QW0.8212:INT;	(* +/- xxxx W *)
	SRV_EP_wattmeter09_var AT %QW0.8216:INT;	(* +/- xxxx var *)
	SRV_EP_wattmeter09_VA AT %QW0.8220:INT;	(* +/- xxxx VA *)
	SRV_EP_wattmeter09_kWh AT %QD0.8224:DINT;	(* xxxxxxxxx.x +kWh *)
	SRV_EP_wattmeter10_W AT %QW0.8228:INT;	(* +/- xxxx W *)
	SRV_EP_wattmeter10_var AT %QW0.8232:INT;	(* +/- xxxx var *)
	SRV_EP_wattmeter10_VA AT %QW0.8236:INT;	(* +/- xxxx VA *)
	SRV_EP_wattmeter10_kWh AT %QD0.8240:DINT;	(* xxxxxxxxx.x +kWh *)
	SRV_EP_BlackoutDetected AT %QX0.8244.0:BOOL;
	SRV_EP_OverloadDetected AT %QX0.8248.0:BOOL;
	SRV_EP_enabled_relays AT %QW0.8252:INT;	(* 0 .. 8 *)
	SRV_EP_relay_A AT %QX0.8256.0:BOOL;
	SRV_EP_relay_B AT %QX0.8260.0:BOOL;
	SRV_EP_relay_C AT %QX0.8264.0:BOOL;
	SRV_EP_relay_D AT %QX0.8268.0:BOOL;
	SRV_EP_relay_E AT %QX0.8272.0:BOOL;
	SRV_EP_relay_F AT %QX0.8276.0:BOOL;
	SRV_EP_relay_G AT %QX0.8280.0:BOOL;
	SRV_EP_relay_H AT %QX0.8284.0:BOOL;
	SRV_EP_overload_W AT %QW0.8288:UINT;
	SRV_EP_max_assigned_W AT %QW0.8292:UINT;
	SRV_EP_tic_in_tac AT %QW0.8296:UINT;
	SRV_EP_requested_W AT %QW0.8300:UINT;
	SRV_EP_T1_assigned_W AT %QW0.8304:UINT;
	SRV_EP_T2_assigned_W AT %QW0.8308:UINT;
	SRV_EP_T3_assigned_W AT %QW0.8312:UINT;
	SRV_EP_T4_assigned_W AT %QW0.8316:UINT;
	SRV_EP_T5_assigned_W AT %QW0.8320:UINT;
	SRV_EP_T6_assigned_W AT %QW0.8324:UINT;
	SRV_EP_assigned_W AT %QW0.8328:UINT;
	SRV_EP_control_type AT %QW0.8332:UINT;
	SRV_T1_heartbeat AT %QW0.8400:UINT;	(* TCPS_STATUS NODE_09_STATUS *)
	SRV_T1_enabled_sensors AT %QW0.8404:INT;
	SRV_T1_temperature AT %QW0.8408:INT;
	SRV_T1_temperature_bis AT %QW0.8412:INT;
	SRV_T1_temperature_ext AT %QW0.8416:INT;
	SRV_T1_humidity AT %QW0.8420:INT;
	SRV_T1_humidity_bis AT %QW0.8424:INT;
	SRV_T1_humidity_ext AT %QW0.8428:INT;
	SRV_T1_temperature_setpoint AT %QW0.8432:INT;
	SRV_T1_humidity_setpoint AT %QW0.8436:INT;
	SRV_T1_enabled_lamps AT %QW0.8440:UINT;
	SRV_T1_lamp_1 AT %QX0.8444.0:BOOL;
	SRV_T1_lamp_2 AT %QX0.8448.0:BOOL;
	SRV_T1_lamp_3 AT %QX0.8452.0:BOOL;
	SRV_T1_lamp_4 AT %QX0.8456.0:BOOL;
	SRV_T1_lamp_5 AT %QX0.8460.0:BOOL;
	SRV_T1_max_request_W AT %QW0.8464:UINT;
	SRV_T1_heating AT %QX0.8468.0:BOOL;
	SRV_T1_nighttime AT %QX0.8472.0:BOOL;
	SRV_T1_heating_status AT %QW0.8476:INT;
	SRV_T1_heating_timer AT %QW0.8480:INT;
	SRV_T1_sunrise AT %QW0.8484:UINT;
	SRV_T1_sunset AT %QW0.8488:UINT;	(* hh * 100 + mm *)
	SRV_T1_temperature_setpoint_nt AT %QW0.8492:INT;	(* hh * 100 + mm *)
	SRV_T1_humidity_setpoint_nt AT %QW0.8496:INT;
	SRV_T1_lamp_feedback_1 AT %QX0.8500.0:BOOL;
	SRV_T1_lamp_feedback_2 AT %QX0.8504.0:BOOL;
	SRV_T1_lamp_feedback_3 AT %QX0.8508.0:BOOL;
	SRV_T1_lamp_feedback_4 AT %QX0.8512.0:BOOL;
	SRV_T1_lamp_feedback_5 AT %QX0.8516.0:BOOL;
	SRV_T1_requested_W AT %QW0.8520:UINT;
	SRV_T1_control_type AT %QW0.8524:UINT;
	SRV_T1_daily_heating_s AT %QD0.8528:UDINT;
	SRV_T1_monthly_heating_s AT %QD0.8532:UDINT;
	SRV_T2_heartbeat AT %QW0.8600:UINT;	(* TCPS_STATUS NODE_09_STATUS *)
	SRV_T2_enabled_sensors AT %QW0.8604:INT;
	SRV_T2_temperature AT %QW0.8608:INT;
	SRV_T2_temperature_bis AT %QW0.8612:INT;
	SRV_T2_temperature_ext AT %QW0.8616:INT;
	SRV_T2_humidity AT %QW0.8620:INT;
	SRV_T2_humidity_bis AT %QW0.8624:INT;
	SRV_T2_humidity_ext AT %QW0.8628:INT;
	SRV_T2_temperature_setpoint AT %QW0.8632:INT;
	SRV_T2_humidity_setpoint AT %QW0.8636:INT;
	SRV_T2_enabled_lamps AT %QW0.8640:UINT;
	SRV_T2_lamp_1 AT %QX0.8644.0:BOOL;
	SRV_T2_lamp_2 AT %QX0.8648.0:BOOL;
	SRV_T2_lamp_3 AT %QX0.8652.0:BOOL;
	SRV_T2_lamp_4 AT %QX0.8656.0:BOOL;
	SRV_T2_lamp_5 AT %QX0.8660.0:BOOL;
	SRV_T2_max_request_W AT %QW0.8664:UINT;
	SRV_T2_heating AT %QX0.8668.0:BOOL;
	SRV_T2_nighttime AT %QX0.8672.0:BOOL;
	SRV_T2_heating_status AT %QW0.8676:INT;
	SRV_T2_heating_timer AT %QW0.8680:INT;
	SRV_T2_sunrise AT %QW0.8684:UINT;	(* hh * 100 + mm *)
	SRV_T2_sunset AT %QW0.8688:UINT;	(* hh * 100 + mm *)
	SRV_T2_temperature_setpoint_nt AT %QW0.8692:INT;
	SRV_T2_humidity_setpoint_nt AT %QW0.8696:INT;
	SRV_T2_lamp_feedback_1 AT %QX0.8700.0:BOOL;
	SRV_T2_lamp_feedback_2 AT %QX0.8704.0:BOOL;
	SRV_T2_lamp_feedback_3 AT %QX0.8708.0:BOOL;
	SRV_T2_lamp_feedback_4 AT %QX0.8712.0:BOOL;
	SRV_T2_lamp_feedback_5 AT %QX0.8716.0:BOOL;
	SRV_T2_requested_W AT %QW0.8720:UINT;
	SRV_T2_control_type AT %QW0.8724:UINT;
	SRV_T2_daily_heating_s AT %QD0.8728:UDINT;
	SRV_T2_monthly_heating_s AT %QD0.8732:UDINT;
	SRV_T3_heartbeat AT %QW0.8800:UINT;	(* TCPS_STATUS NODE_09_STATUS *)
	SRV_T3_enabled_sensors AT %QW0.8804:INT;
	SRV_T3_temperature AT %QW0.8808:INT;
	SRV_T3_temperature_bis AT %QW0.8812:INT;
	SRV_T3_temperature_ext AT %QW0.8816:INT;
	SRV_T3_humidity AT %QW0.8820:INT;
	SRV_T3_humidity_bis AT %QW0.8824:INT;
	SRV_T3_humidity_ext AT %QW0.8828:INT;
	SRV_T3_temperature_setpoint AT %QW0.8832:INT;
	SRV_T3_humidity_setpoint AT %QW0.8836:INT;
	SRV_T3_enabled_lamps AT %QW0.8840:UINT;
	SRV_T3_lamp_1 AT %QX0.8844.0:BOOL;
	SRV_T3_lamp_2 AT %QX0.8848.0:BOOL;
	SRV_T3_lamp_3 AT %QX0.8852.0:BOOL;
	SRV_T3_lamp_4 AT %QX0.8856.0:BOOL;
	SRV_T3_lamp_5 AT %QX0.8860.0:BOOL;
	SRV_T3_max_request_W AT %QW0.8864:UINT;
	SRV_T3_heating AT %QX0.8868.0:BOOL;
	SRV_T3_nighttime AT %QX0.8872.0:BOOL;
	SRV_T3_heating_status AT %QW0.8876:INT;
	SRV_T3_heating_timer AT %QW0.8880:INT;
	SRV_T3_sunrise AT %QW0.8884:UINT;	(* hh * 100 + mm *)
	SRV_T3_sunset AT %QW0.8888:UINT;	(* hh * 100 + mm *)
	SRV_T3_temperature_setpoint_nt AT %QW0.8892:INT;
	SRV_T3_humidity_setpoint_nt AT %QW0.8896:INT;
	SRV_T3_lamp_feedback_1 AT %QX0.8900.0:BOOL;
	SRV_T3_lamp_feedback_2 AT %QX0.8904.0:BOOL;
	SRV_T3_lamp_feedback_3 AT %QX0.8908.0:BOOL;
	SRV_T3_lamp_feedback_4 AT %QX0.8912.0:BOOL;
	SRV_T3_lamp_feedback_5 AT %QX0.8916.0:BOOL;
	SRV_T3_requested_W AT %QW0.8920:UINT;
	SRV_T3_control_type AT %QW0.8924:UINT;
	SRV_T3_daily_heating_s AT %QD0.8928:UDINT;
	SRV_T3_monthly_heating_s AT %QD0.8932:UDINT;
	SRV_T4_heartbeat AT %QW0.9000:UINT;	(* TCPS_STATUS NODE_09_STATUS *)
	SRV_T4_enabled_sensors AT %QW0.9004:INT;
	SRV_T4_temperature AT %QW0.9008:INT;
	SRV_T4_temperature_bis AT %QW0.9012:INT;
	SRV_T4_temperature_ext AT %QW0.9016:INT;
	SRV_T4_humidity AT %QW0.9020:INT;
	SRV_T4_humidity_bis AT %QW0.9024:INT;
	SRV_T4_humidity_ext AT %QW0.9028:INT;
	SRV_T4_temperature_setpoint AT %QW0.9032:INT;
	SRV_T4_humidity_setpoint AT %QW0.9036:INT;
	SRV_T4_enabled_lamps AT %QW0.9040:UINT;
	SRV_T4_lamp_1 AT %QX0.9044.0:BOOL;
	SRV_T4_lamp_2 AT %QX0.9048.0:BOOL;
	SRV_T4_lamp_3 AT %QX0.9052.0:BOOL;
	SRV_T4_lamp_4 AT %QX0.9056.0:BOOL;
	SRV_T4_lamp_5 AT %QX0.9060.0:BOOL;
	SRV_T4_max_request_W AT %QW0.9064:UINT;
	SRV_T4_heating AT %QX0.9068.0:BOOL;
	SRV_T4_nighttime AT %QX0.9072.0:BOOL;
	SRV_T4_heating_status AT %QW0.9076:INT;
	SRV_T4_heating_timer AT %QW0.9080:INT;
	SRV_T4_sunrise AT %QW0.9084:UINT;	(* hh * 100 + mm *)
	SRV_T4_sunset AT %QW0.9088:UINT;	(* hh * 100 + mm *)
	SRV_T4_temperature_setpoint_nt AT %QW0.9092:INT;
	SRV_T4_humidity_setpoint_nt AT %QW0.9096:INT;
	SRV_T4_lamp_feedback_1 AT %QX0.9100.0:BOOL;
	SRV_T4_lamp_feedback_2 AT %QX0.9104.0:BOOL;
	SRV_T4_lamp_feedback_3 AT %QX0.9108.0:BOOL;
	SRV_T4_lamp_feedback_4 AT %QX0.9112.0:BOOL;
	SRV_T4_lamp_feedback_5 AT %QX0.9116.0:BOOL;
	SRV_T4_requested_W AT %QW0.9120:UINT;
	SRV_T4_control_type AT %QW0.9124:UINT;
	SRV_T4_daily_heating_s AT %QD0.9128:UDINT;
	SRV_T4_monthly_heating_s AT %QD0.9132:UDINT;
	SRV_T5_heartbeat AT %QW0.9200:UINT;	(* TCPS_STATUS NODE_09_STATUS *)
	SRV_T5_enabled_sensors AT %QW0.9204:INT;
	SRV_T5_temperature AT %QW0.9208:INT;
	SRV_T5_temperature_bis AT %QW0.9212:INT;
	SRV_T5_temperature_ext AT %QW0.9216:INT;
	SRV_T5_humidity AT %QW0.9220:INT;
	SRV_T5_humidity_bis AT %QW0.9224:INT;
	SRV_T5_humidity_ext AT %QW0.9228:INT;
	SRV_T5_temperature_setpoint AT %QW0.9232:INT;
	SRV_T5_humidity_setpoint AT %QW0.9236:INT;
	SRV_T5_enabled_lamps AT %QW0.9240:UINT;
	SRV_T5_lamp_1 AT %QX0.9244.0:BOOL;
	SRV_T5_lamp_2 AT %QX0.9248.0:BOOL;
	SRV_T5_lamp_3 AT %QX0.9252.0:BOOL;
	SRV_T5_lamp_4 AT %QX0.9256.0:BOOL;
	SRV_T5_lamp_5 AT %QX0.9260.0:BOOL;
	SRV_T5_max_request_W AT %QW0.9264:UINT;
	SRV_T5_heating AT %QX0.9268.0:BOOL;
	SRV_T5_nighttime AT %QX0.9272.0:BOOL;
	SRV_T5_heating_status AT %QW0.9276:INT;
	SRV_T5_heating_timer AT %QW0.9280:INT;
	SRV_T5_sunrise AT %QW0.9284:UINT;	(* hh * 100 + mm *)
	SRV_T5_sunset AT %QW0.9288:UINT;	(* hh * 100 + mm *)
	SRV_T5_temperature_setpoint_nt AT %QW0.9292:INT;
	SRV_T5_humidity_setpoint_nt AT %QW0.9296:INT;
	SRV_T5_lamp_feedback_1 AT %QX0.9300.0:BOOL;
	SRV_T5_lamp_feedback_2 AT %QX0.9304.0:BOOL;
	SRV_T5_lamp_feedback_3 AT %QX0.9308.0:BOOL;
	SRV_T5_lamp_feedback_4 AT %QX0.9312.0:BOOL;
	SRV_T5_lamp_feedback_5 AT %QX0.9316.0:BOOL;
	SRV_T5_requested_W AT %QW0.9320:UINT;
	SRV_T5_control_type AT %QW0.9324:UINT;
	SRV_T5_daily_heating_s AT %QD0.9328:UDINT;
	SRV_T5_monthly_heating_s AT %QD0.9332:UDINT;
	SRV_T6_heartbeat AT %QW0.9400:UINT;	(* TCPS_STATUS NODE_09_STATUS *)
	SRV_T6_enabled_sensors AT %QW0.9404:INT;
	SRV_T6_temperature AT %QW0.9408:INT;
	SRV_T6_temperature_bis AT %QW0.9412:INT;
	SRV_T6_temperature_ext AT %QW0.9416:INT;
	SRV_T6_humidity AT %QW0.9420:INT;
	SRV_T6_humidity_bis AT %QW0.9424:INT;
	SRV_T6_humidity_ext AT %QW0.9428:INT;
	SRV_T6_temperature_setpoint AT %QW0.9432:INT;
	SRV_T6_humidity_setpoint AT %QW0.9436:INT;
	SRV_T6_enabled_lamps AT %QW0.9440:UINT;
	SRV_T6_lamp_1 AT %QX0.9444.0:BOOL;
	SRV_T6_lamp_2 AT %QX0.9448.0:BOOL;
	SRV_T6_lamp_3 AT %QX0.9452.0:BOOL;
	SRV_T6_lamp_4 AT %QX0.9456.0:BOOL;
	SRV_T6_lamp_5 AT %QX0.9460.0:BOOL;
	SRV_T6_max_request_W AT %QW0.9464:UINT;
	SRV_T6_heating AT %QX0.9468.0:BOOL;
	SRV_T6_nighttime AT %QX0.9472.0:BOOL;
	SRV_T6_heating_status AT %QW0.9476:INT;
	SRV_T6_heating_timer AT %QW0.9480:INT;
	SRV_T6_sunrise AT %QW0.9484:UINT;	(* hh * 100 + mm *)
	SRV_T6_sunset AT %QW0.9488:UINT;	(* hh * 100 + mm *)
	SRV_T6_temperature_setpoint_nt AT %QW0.9492:INT;
	SRV_T6_humidity_setpoint_nt AT %QW0.9496:INT;
	SRV_T6_lamp_feedback_1 AT %QX0.9500.0:BOOL;
	SRV_T6_lamp_feedback_2 AT %QX0.9504.0:BOOL;
	SRV_T6_lamp_feedback_3 AT %QX0.9508.0:BOOL;
	SRV_T6_lamp_feedback_4 AT %QX0.9512.0:BOOL;
	SRV_T6_lamp_feedback_5 AT %QX0.9516.0:BOOL;
	SRV_T6_requested_W AT %QW0.9520:UINT;
	SRV_T6_control_type AT %QW0.9524:UINT;
	SRV_T6_daily_heating_s AT %QD0.9528:UDINT;
	SRV_T6_monthly_heating_s AT %QD0.9532:UDINT;
	SRV_BA_heartbeat AT %QW0.10800:UINT;	(* TCP7_STATUS NODE_08_STATUS *)
	SRV_BA_enabled_sensors AT %QW0.10804:UINT;	(* 0, 8, 16, 24, 32 *)
	SRV_BA_status AT %QW0.10808:UINT;	(* ZERO, OFF, ARMED, ENABLED, RINGING, MUTED, TESTING *)
	SRV_BA_config_index AT %QW0.10812:UINT;	(* 0 1 2 3 *)
	SRV_BA_config_mask AT %QD0.10816:UDINT;	(* 32 bit mask *)
	SRV_BA_led_green AT %QX0.10820.0:BOOL;	(* ARMED(blinking), ENABLED, RINGING, MUTED *)
	SRV_BA_led_red AT %QX0.10824.0:BOOL;	(* ARMED(if NG), RINGING(blinking), MUTED *)
	SRV_BA_led_yellow1 AT %QX0.10828.0:BOOL;	(* NIGHTIME, EVERYTHING *)
	SRV_BA_led_yellow2 AT %QX0.10832.0:BOOL;	(* DAYTIME, EVERYTHING *)
	SRV_BA_siren AT %QX0.10836.0:BOOL;	(* HPA *)
	SRV_BA_relay_A AT %QX0.10840.0:BOOL;
	SRV_BA_relay_B AT %QX0.10844.0:BOOL;
	SRV_BA_relay_C AT %QX0.10848.0:BOOL;
	SRV_BA_input_9 AT %QX0.10852.0:BOOL;
	SRV_BA_input_10 AT %QX0.10856.0:BOOL;
	SRV_BA_input_11 AT %QX0.10860.0:BOOL;
	SRV_BA_input_12 AT %QX0.10864.0:BOOL;
	SRV_BA_BlackoutDetected AT %QX0.10868.0:BOOL;
	SRV_BA_command AT %QD0.10872:UDINT;	(* NONE, ARM, NOTHING, DAYTIME, NIGHTIME, EVERYTHING, ENABLE, DISABLE, ACK, TEST *)
	SRV_BA_OK_1 AT %QW0.10876:UINT;
	SRV_BA_OK_2 AT %QW0.10880:UINT;
	SRV_BA_OK_3 AT %QW0.10884:UINT;
	SRV_BA_OK_4 AT %QW0.10888:UINT;
	SRV_BA_OK_5 AT %QW0.10892:UINT;
	SRV_BA_OK_6 AT %QW0.10896:UINT;
	SRV_BA_OK_7 AT %QW0.10900:UINT;
	SRV_BA_OK_8 AT %QW0.10904:UINT;
	SRV_BA_OK_9 AT %QW0.10908:UINT;
	SRV_BA_OK_10 AT %QW0.10912:UINT;
	SRV_BA_OK_11 AT %QW0.10916:UINT;
	SRV_BA_OK_12 AT %QW0.10920:UINT;
	SRV_BA_OK_13 AT %QW0.10924:UINT;
	SRV_BA_OK_14 AT %QW0.10928:UINT;
	SRV_BA_OK_15 AT %QW0.10932:UINT;
	SRV_BA_OK_16 AT %QW0.10936:UINT;
	SRV_BA_OK_17 AT %QW0.10940:UINT;
	SRV_BA_OK_18 AT %QW0.10944:UINT;
	SRV_BA_OK_19 AT %QW0.10948:UINT;
	SRV_BA_OK_20 AT %QW0.10952:UINT;
	SRV_BA_OK_21 AT %QW0.10956:UINT;
	SRV_BA_OK_22 AT %QW0.10960:UINT;
	SRV_BA_OK_23 AT %QW0.10964:UINT;
	SRV_BA_OK_24 AT %QW0.10968:UINT;
	SRV_BA_OK_25 AT %QW0.10972:UINT;
	SRV_BA_OK_26 AT %QW0.10976:UINT;
	SRV_BA_OK_27 AT %QW0.10980:UINT;
	SRV_BA_OK_28 AT %QW0.10984:UINT;
	SRV_BA_OK_29 AT %QW0.10988:UINT;
	SRV_BA_OK_30 AT %QW0.10992:UINT;
	SRV_BA_OK_31 AT %QW0.10996:UINT;
	SRV_BA_OK_32 AT %QW0.11000:UINT;
	SRV_BA_control_type AT %QW0.11004:UINT;
	PLC_EP_wattmeters_ok AT %QW0.12016:UINT;	(* bit mask (node status) *)
	PLC_EP_wattmeter_M_W AT %QW0.12020:INT;	(* +/- xxxx W *)
	PLC_EP_wattmeter_M_var AT %QW0.12024:INT;	(* +/- xxxx var *)
	PLC_EP_wattmeter_M_VA AT %QW0.12028:INT;	(* +/- xxxx VA *)
	PLC_EP_wattmeter_M_pf AT %QW0.12032:INT;	(* +/- x.xxx *)
	PLC_EP_wattmeter_M_Hz AT %QW0.12036:INT;	(* xxx.xx Hz *)
	PLC_EP_wattmeter_M_V AT %QW0.12040:INT;	(* xxx.xx V *)
	PLC_EP_wattmeter_M_1_A AT %QW0.12044:INT;	(* xx.xxx A *)
	PLC_EP_wattmeter_M_2_A AT %QW0.12048:INT;	(* xx.xxx A *)
	PLC_EP_wattmeter_M_3_A AT %QW0.12052:INT;	(* xx.xxx A *)
	PLC_EP_wattmeter_M_A AT %QW0.12056:INT;	(* xx.xxx A *)
	PLC_EP_wattmeter_M_kWh AT %QD0.12060:DINT;	(* xxxxxxxxx.x +kWh *)
	PLC_EP_wattmeter_M_e_kWh AT %QD0.12064:DINT;	(* xxxxxxxxx.x -kWh *)
	PLC_EP_wattmeter_F_W AT %QW0.12068:INT;	(* +/- xxxx W *)
	PLC_EP_wattmeter_F_var AT %QW0.12072:INT;	(* +/- xxxx var *)
	PLC_EP_wattmeter_F_VA AT %QW0.12076:INT;	(* +/- xxxx VA *)
	PLC_EP_wattmeter_F_pf AT %QW0.12080:INT;	(* +/- x.xxx *)
	PLC_EP_wattmeter_F_Hz AT %QW0.12084:INT;	(* xxx.xx Hz *)
	PLC_EP_wattmeter_F_V AT %QW0.12088:INT;	(* xxx.xx V *)
	PLC_EP_wattmeter_F_1_A AT %QW0.12092:INT;	(* xx.xxx A *)
	PLC_EP_wattmeter_F_2_A AT %QW0.12096:INT;	(* xx.xxx A *)
	PLC_EP_wattmeter_F_3_A AT %QW0.12100:INT;	(* xx.xxx A *)
	PLC_EP_wattmeter_F_A AT %QW0.12104:INT;	(* xx.xxx A *)
	PLC_EP_wattmeter_F_kWh AT %QD0.12108:DINT;	(* xxxxxxxxx.x +kWh *)
	PLC_EP_wattmeter_F_e_kWh AT %QD0.12112:DINT;	(* xxxxxxxxx.x -kWh *)
	PLC_EP_wattmeter01_W AT %QW0.12116:INT;	(* +/- xxxx W *)
	PLC_EP_wattmeter01_var AT %QW0.12120:INT;	(* +/- xxxx var *)
	PLC_EP_wattmeter01_VA AT %QW0.12124:INT;	(* +/- xxxx VA *)
	PLC_EP_wattmeter01_kWh AT %QD0.12128:DINT;	(* xxxxxxxxx.x kWh *)
	PLC_EP_wattmeter02_W AT %QW0.12132:INT;	(* +/- xxxx W *)
	PLC_EP_wattmeter02_var AT %QW0.12136:INT;	(* +/- xxxx var *)
	PLC_EP_wattmeter02_VA AT %QW0.12140:INT;	(* +/- xxxx VA *)
	PLC_EP_wattmeter02_kWh AT %QD0.12144:DINT;	(* xxxxxxxxx.x kWh *)
	PLC_EP_wattmeter03_W AT %QW0.12148:INT;	(* +/- xxxx W *)
	PLC_EP_wattmeter03_var AT %QW0.12152:INT;	(* +/- xxxx var *)
	PLC_EP_wattmeter03_VA AT %QW0.12156:INT;	(* +/- xxxx VA *)
	PLC_EP_wattmeter03_kWh AT %QD0.12160:DINT;	(* xxxxxxxxx.x kWh *)
	PLC_EP_wattmeter04_W AT %QW0.12164:INT;	(* +/- xxxx W *)
	PLC_EP_wattmeter04_var AT %QW0.12168:INT;	(* +/- xxxx var *)
	PLC_EP_wattmeter04_VA AT %QW0.12172:INT;	(* +/- xxxx VA *)
	PLC_EP_wattmeter04_kWh AT %QD0.12176:DINT;	(* xxxxxxxxx.x kWh *)
	PLC_EP_wattmeter05_W AT %QW0.12180:INT;	(* +/- xxxx W *)
	PLC_EP_wattmeter05_var AT %QW0.12184:INT;	(* +/- xxxx var *)
	PLC_EP_wattmeter05_VA AT %QW0.12188:INT;	(* +/- xxxx VA *)
	PLC_EP_wattmeter05_kWh AT %QD0.12192:DINT;	(* xxxxxxxxx.x kWh *)
	PLC_EP_wattmeter06_W AT %QW0.12196:INT;	(* +/- xxxx W *)
	PLC_EP_wattmeter06_var AT %QW0.12200:INT;	(* +/- xxxx var *)
	PLC_EP_wattmeter06_VA AT %QW0.12204:INT;	(* +/- xxxx VA *)
	PLC_EP_wattmeter06_kWh AT %QD0.12208:DINT;	(* xxxxxxxxx.x kWh *)
	PLC_EP_wattmeter07_W AT %QW0.12212:INT;	(* +/- xxxx W *)
	PLC_EP_wattmeter07_var AT %QW0.12216:INT;	(* +/- xxxx var *)
	PLC_EP_wattmeter07_VA AT %QW0.12220:INT;	(* +/- xxxx VA *)
	PLC_EP_wattmeter07_kWh AT %QD0.12224:DINT;	(* xxxxxxxxx.x kWh *)
	PLC_EP_wattmeter08_W AT %QW0.12228:INT;	(* +/- xxxx W *)
	PLC_EP_wattmeter08_var AT %QW0.12232:INT;	(* +/- xxxx var *)
	PLC_EP_wattmeter08_VA AT %QW0.12236:INT;	(* +/- xxxx VA *)
	PLC_EP_wattmeter08_kWh AT %QD0.12240:DINT;	(* xxxxxxxxx.x kWh *)
	PLC_EP_wattmeter09_W AT %QW0.12244:INT;	(* +/- xxxx W *)
	PLC_EP_wattmeter09_var AT %QW0.12248:INT;	(* +/- xxxx var *)
	PLC_EP_wattmeter09_VA AT %QW0.12252:INT;	(* +/- xxxx VA *)
	PLC_EP_wattmeter09_kWh AT %QD0.12256:DINT;	(* xxxxxxxxx.x kWh *)
	PLC_EP_wattmeter10_W AT %QW0.12260:INT;	(* +/- xxxx W *)
	PLC_EP_wattmeter10_var AT %QW0.12264:INT;	(* +/- xxxx var *)
	PLC_EP_wattmeter10_VA AT %QW0.12268:INT;	(* +/- xxxx VA *)
	PLC_EP_wattmeter10_kWh AT %QD0.12272:DINT;	(* xxxxxxxxx.x kWh *)
	PLC_EP_relay_A AT %QX0.12276.0:BOOL;
	PLC_EP_relay_B AT %QX0.12280.0:BOOL;
	PLC_EP_relay_C AT %QX0.12284.0:BOOL;
	PLC_EP_relay_D AT %QX0.12288.0:BOOL;
	PLC_EP_relay_E AT %QX0.12292.0:BOOL;
	PLC_EP_relay_F AT %QX0.12296.0:BOOL;
	PLC_EP_relay_G AT %QX0.12300.0:BOOL;
	PLC_EP_relay_H AT %QX0.12304.0:BOOL;
	PLC_EP_tic_in_tac AT %QW0.12308:UINT;
	PLC_T1_requested_W AT %QW0.12312:UINT;
	PLC_T2_requested_W AT %QW0.12316:UINT;
	PLC_T3_requested_W AT %QW0.12320:UINT;
	PLC_T4_requested_W AT %QW0.12324:UINT;
	PLC_T5_requested_W AT %QW0.12328:UINT;
	PLC_T6_requested_W AT %QW0.12332:UINT;
	PLC_EP_requested_W AT %QW0.12336:UINT;	(* total requested W *)
	PLC_EP_T1_assigned_W AT %QW0.12340:UINT;
	PLC_EP_T2_assigned_W AT %QW0.12344:UINT;
	PLC_EP_T3_assigned_W AT %QW0.12348:UINT;
	PLC_EP_T4_assigned_W AT %QW0.12352:UINT;
	PLC_EP_T5_assigned_W AT %QW0.12356:UINT;
	PLC_EP_T6_assigned_W AT %QW0.12360:UINT;
	PLC_EP_assigned_W AT %QW0.12364:UINT;	(* total assigned W *)
	PLC_EP_control_type AT %QW0.12368:UINT;
	PLC_T1_temperature AT %QW0.12400:INT;
	PLC_T1_temperature_bis AT %QW0.12404:INT;
	PLC_T1_temperature_ext AT %QW0.12408:INT;
	PLC_T1_humidity AT %QW0.12412:INT;
	PLC_T1_humidity_bis AT %QW0.12416:INT;
	PLC_T1_humidity_ext AT %QW0.12420:INT;
	PLC_T1_lamp_1 AT %QX0.12424.0:BOOL;
	PLC_T1_lamp_2 AT %QX0.12428.0:BOOL;
	PLC_T1_lamp_3 AT %QX0.12432.0:BOOL;
	PLC_T1_lamp_4 AT %QX0.12436.0:BOOL;
	PLC_T1_lamp_5 AT %QX0.12440.0:BOOL;
	PLC_T1_sunrise AT %QW0.12444:UINT;	(* hh * 100 + mm *)
	PLC_T1_sunset AT %QW0.12448:UINT;	(* hh * 100 + mm *)
	PLC_T1_heating AT %QX0.12452.0:BOOL;
	PLC_T1_nighttime AT %QX0.12456.0:BOOL;
	PLC_T1_heating_timer AT %QW0.12460:INT;
	PLC_T1_lamp_feedback_1 AT %QX0.12464.0:BOOL;
	PLC_T1_lamp_feedback_2 AT %QX0.12468.0:BOOL;
	PLC_T1_lamp_feedback_3 AT %QX0.12472.0:BOOL;
	PLC_T1_lamp_feedback_4 AT %QX0.12476.0:BOOL;
	PLC_T1_lamp_feedback_5 AT %QX0.12480.0:BOOL;
	PLC_T1_control_type AT %QW0.12484:UINT;
	PLC_T2_temperature AT %QW0.12600:INT;
	PLC_T2_temperature_bis AT %QW0.12604:INT;
	PLC_T2_temperature_ext AT %QW0.12608:INT;
	PLC_T2_humidity AT %QW0.12612:INT;
	PLC_T2_humidity_bis AT %QW0.12616:INT;
	PLC_T2_humidity_ext AT %QW0.12620:INT;
	PLC_T2_lamp_1 AT %QX0.12624.0:BOOL;
	PLC_T2_lamp_2 AT %QX0.12628.0:BOOL;
	PLC_T2_lamp_3 AT %QX0.12632.0:BOOL;
	PLC_T2_lamp_4 AT %QX0.12636.0:BOOL;
	PLC_T2_lamp_5 AT %QX0.12640.0:BOOL;
	PLC_T2_sunrise AT %QW0.12644:UINT;	(* hh * 100 + mm *)
	PLC_T2_sunset AT %QW0.12648:UINT;	(* hh * 100 + mm *)
	PLC_T2_heating AT %QX0.12652.0:BOOL;
	PLC_T2_nighttime AT %QX0.12656.0:BOOL;
	PLC_T2_heating_timer AT %QW0.12660:INT;
	PLC_T2_lamp_feedback_1 AT %QX0.12664.0:BOOL;
	PLC_T2_lamp_feedback_2 AT %QX0.12668.0:BOOL;
	PLC_T2_lamp_feedback_3 AT %QX0.12672.0:BOOL;
	PLC_T2_lamp_feedback_4 AT %QX0.12676.0:BOOL;
	PLC_T2_lamp_feedback_5 AT %QX0.12680.0:BOOL;
	PLC_T2_control_type AT %QW0.12684:UINT;
	PLC_T3_temperature AT %QW0.12800:INT;
	PLC_T3_temperature_bis AT %QW0.12804:INT;
	PLC_T3_temperature_ext AT %QW0.12808:INT;
	PLC_T3_humidity AT %QW0.12812:INT;
	PLC_T3_humidity_bis AT %QW0.12816:INT;
	PLC_T3_humidity_ext AT %QW0.12820:INT;
	PLC_T3_lamp_1 AT %QX0.12824.0:BOOL;
	PLC_T3_lamp_2 AT %QX0.12828.0:BOOL;
	PLC_T3_lamp_3 AT %QX0.12832.0:BOOL;
	PLC_T3_lamp_4 AT %QX0.12836.0:BOOL;
	PLC_T3_lamp_5 AT %QX0.12840.0:BOOL;
	PLC_T3_sunrise AT %QW0.12844:UINT;	(* hh * 100 + mm *)
	PLC_T3_sunset AT %QW0.12848:UINT;	(* hh * 100 + mm *)
	PLC_T3_heating AT %QX0.12852.0:BOOL;
	PLC_T3_nighttime AT %QX0.12856.0:BOOL;
	PLC_T3_heating_timer AT %QW0.12860:INT;
	PLC_T3_lamp_feedback_1 AT %QX0.12864.0:BOOL;
	PLC_T3_lamp_feedback_2 AT %QX0.12868.0:BOOL;
	PLC_T3_lamp_feedback_3 AT %QX0.12872.0:BOOL;
	PLC_T3_lamp_feedback_4 AT %QX0.12876.0:BOOL;
	PLC_T3_lamp_feedback_5 AT %QX0.12880.0:BOOL;
	PLC_T3_control_type AT %QW0.12884:UINT;
	PLC_T4_temperature AT %QW0.13000:INT;
	PLC_T4_temperature_bis AT %QW0.13004:INT;
	PLC_T4_temperature_ext AT %QW0.13008:INT;
	PLC_T4_humidity AT %QW0.13012:INT;
	PLC_T4_humidity_bis AT %QW0.13016:INT;
	PLC_T4_humidity_ext AT %QW0.13020:INT;
	PLC_T4_lamp_1 AT %QX0.13024.0:BOOL;
	PLC_T4_lamp_2 AT %QX0.13028.0:BOOL;
	PLC_T4_lamp_3 AT %QX0.13032.0:BOOL;
	PLC_T4_lamp_4 AT %QX0.13036.0:BOOL;
	PLC_T4_lamp_5 AT %QX0.13040.0:BOOL;
	PLC_T4_sunrise AT %QW0.13044:UINT;	(* hh * 100 + mm *)
	PLC_T4_sunset AT %QW0.13048:UINT;	(* hh * 100 + mm *)
	PLC_T4_heating AT %QX0.13052.0:BOOL;
	PLC_T4_nighttime AT %QX0.13056.0:BOOL;
	PLC_T4_heating_timer AT %QW0.13060:INT;
	PLC_T4_lamp_feedback_1 AT %QX0.13064.0:BOOL;
	PLC_T4_lamp_feedback_2 AT %QX0.13068.0:BOOL;
	PLC_T4_lamp_feedback_3 AT %QX0.13072.0:BOOL;
	PLC_T4_lamp_feedback_4 AT %QX0.13076.0:BOOL;
	PLC_T4_lamp_feedback_5 AT %QX0.13080.0:BOOL;
	PLC_T4_control_type AT %QW0.13084:UINT;
	PLC_T5_temperature AT %QW0.13200:INT;
	PLC_T5_temperature_bis AT %QW0.13204:INT;
	PLC_T5_temperature_ext AT %QW0.13208:INT;
	PLC_T5_humidity AT %QW0.13212:INT;
	PLC_T5_humidity_bis AT %QW0.13216:INT;
	PLC_T5_humidity_ext AT %QW0.13220:INT;
	PLC_T5_lamp_1 AT %QX0.13224.0:BOOL;
	PLC_T5_lamp_2 AT %QX0.13228.0:BOOL;
	PLC_T5_lamp_3 AT %QX0.13232.0:BOOL;
	PLC_T5_lamp_4 AT %QX0.13236.0:BOOL;
	PLC_T5_lamp_5 AT %QX0.13240.0:BOOL;
	PLC_T5_sunrise AT %QW0.13244:UINT;	(* hh * 100 + mm *)
	PLC_T5_sunset AT %QW0.13248:UINT;	(* hh * 100 + mm *)
	PLC_T5_heating AT %QX0.13252.0:BOOL;
	PLC_T5_nighttime AT %QX0.13256.0:BOOL;
	PLC_T5_heating_timer AT %QW0.13260:INT;
	PLC_T5_lamp_feedback_1 AT %QX0.13264.0:BOOL;
	PLC_T5_lamp_feedback_2 AT %QX0.13268.0:BOOL;
	PLC_T5_lamp_feedback_3 AT %QX0.13272.0:BOOL;
	PLC_T5_lamp_feedback_4 AT %QX0.13276.0:BOOL;
	PLC_T5_lamp_feedback_5 AT %QX0.13280.0:BOOL;
	PLC_T5_control_type AT %QW0.13284:UINT;
	PLC_T6_temperature AT %QW0.13400:INT;
	PLC_T6_temperature_bis AT %QW0.13404:INT;
	PLC_T6_temperature_ext AT %QW0.13408:INT;
	PLC_T6_humidity AT %QW0.13412:INT;
	PLC_T6_humidity_bis AT %QW0.13416:INT;
	PLC_T6_humidity_ext AT %QW0.13420:INT;
	PLC_T6_lamp_1 AT %QX0.13424.0:BOOL;
	PLC_T6_lamp_2 AT %QX0.13428.0:BOOL;
	PLC_T6_lamp_3 AT %QX0.13432.0:BOOL;
	PLC_T6_lamp_4 AT %QX0.13436.0:BOOL;
	PLC_T6_lamp_5 AT %QX0.13440.0:BOOL;
	PLC_T6_sunrise AT %QW0.13444:UINT;	(* hh * 100 + mm *)
	PLC_T6_sunset AT %QW0.13448:UINT;	(* hh * 100 + mm *)
	PLC_T6_heating AT %QX0.13452.0:BOOL;
	PLC_T6_nighttime AT %QX0.13456.0:BOOL;
	PLC_T6_heating_timer AT %QW0.13460:INT;
	PLC_T6_lamp_feedback_1 AT %QX0.13464.0:BOOL;
	PLC_T6_lamp_feedback_2 AT %QX0.13468.0:BOOL;
	PLC_T6_lamp_feedback_3 AT %QX0.13472.0:BOOL;
	PLC_T6_lamp_feedback_4 AT %QX0.13476.0:BOOL;
	PLC_T6_lamp_feedback_5 AT %QX0.13480.0:BOOL;
	PLC_T6_control_type AT %QW0.13484:UINT;
	PLC_BA_led_green AT %QX0.14800.0:BOOL;	(* ARMED(blinking), ENABLED, RINGING, MUTED *)
	PLC_BA_led_red AT %QX0.14804.0:BOOL;	(* ARMED(if NG), RINGING(blinking), MUTED *)
	PLC_BA_led_yellow1 AT %QX0.14808.0:BOOL;	(* NIGHTIME, EVERYTHING *)
	PLC_BA_led_yellow2 AT %QX0.14812.0:BOOL;	(* DAYTIME, EVERYTHING *)
	PLC_BA_siren AT %QX0.14816.0:BOOL;	(* HPA *)
	PLC_BA_relay_A AT %QX0.14820.0:BOOL;
	PLC_BA_relay_B AT %QX0.14824.0:BOOL;
	PLC_BA_relay_C AT %QX0.14828.0:BOOL;
	PLC_BA_input_9 AT %QX0.14832.0:BOOL;
	PLC_BA_input_10 AT %QX0.14836.0:BOOL;
	PLC_BA_input_11 AT %QX0.14840.0:BOOL;
	PLC_BA_input_12 AT %QX0.14844.0:BOOL;
	PLC_BA_command AT %QD0.14848:UDINT;	(* NONE, ARM, NOTHING, DAYTIME, NIGHTIME, EVERYTHING, ENABLE, DISABLE, ACK, TEST *)
	PLC_BA_config_mask AT %QD0.14856:UDINT;
	PLC_BA_DigOut_1 AT %QX0.14876.0:BOOL;
	PLC_BA_DigOut_2 AT %QX0.14880.0:BOOL;
	PLC_BA_DigOut_3 AT %QX0.14884.0:BOOL;
	PLC_BA_DigOut_4 AT %QX0.14888.0:BOOL;
	PLC_BA_DigOut_5 AT %QX0.14892.0:BOOL;
	PLC_BA_DigOut_6 AT %QX0.14896.0:BOOL;
	PLC_BA_DigOut_7 AT %QX0.14900.0:BOOL;
	PLC_BA_DigOut_8 AT %QX0.14904.0:BOOL;
	PLC_BA_DigOut_9 AT %QX0.14908.0:BOOL;
	PLC_BA_DigOut_10 AT %QX0.14912.0:BOOL;
	PLC_BA_DigOut_11 AT %QX0.14916.0:BOOL;
	PLC_BA_DigOut_12 AT %QX0.14920.0:BOOL;
	PLC_BA_DigOut_13 AT %QX0.14924.0:BOOL;
	PLC_BA_DigOut_14 AT %QX0.14928.0:BOOL;
	PLC_BA_DigOut_15 AT %QX0.14932.0:BOOL;
	PLC_BA_DigOut_16 AT %QX0.14936.0:BOOL;
	PLC_BA_DigOut_17 AT %QX0.14940.0:BOOL;
	PLC_BA_DigOut_18 AT %QX0.14944.0:BOOL;
	PLC_BA_DigOut_19 AT %QX0.14948.0:BOOL;
	PLC_BA_DigOut_20 AT %QX0.14952.0:BOOL;
	PLC_BA_DigOut_21 AT %QX0.14956.0:BOOL;
	PLC_BA_DigOut_22 AT %QX0.14960.0:BOOL;
	PLC_BA_DigOut_23 AT %QX0.14964.0:BOOL;
	PLC_BA_DigOut_24 AT %QX0.14968.0:BOOL;
	PLC_BA_DigOut_25 AT %QX0.14972.0:BOOL;
	PLC_BA_DigOut_26 AT %QX0.14976.0:BOOL;
	PLC_BA_DigOut_27 AT %QX0.14980.0:BOOL;
	PLC_BA_DigOut_28 AT %QX0.14984.0:BOOL;
	PLC_BA_DigOut_29 AT %QX0.14988.0:BOOL;
	PLC_BA_DigOut_30 AT %QX0.14992.0:BOOL;
	PLC_BA_DigOut_31 AT %QX0.14996.0:BOOL;
	PLC_BA_DigOut_32 AT %QX0.15000.0:BOOL;
	PLC_BA_DigIn_1 AT %QX0.15004.0:BOOL;
	PLC_BA_DigIn_2 AT %QX0.15008.0:BOOL;
	PLC_BA_DigIn_3 AT %QX0.15012.0:BOOL;
	PLC_BA_DigIn_4 AT %QX0.15016.0:BOOL;
	PLC_BA_DigIn_5 AT %QX0.15020.0:BOOL;
	PLC_BA_DigIn_6 AT %QX0.15024.0:BOOL;
	PLC_BA_DigIn_7 AT %QX0.15028.0:BOOL;
	PLC_BA_DigIn_8 AT %QX0.15032.0:BOOL;
	PLC_BA_DigIn_9 AT %QX0.15036.0:BOOL;
	PLC_BA_DigIn_10 AT %QX0.15040.0:BOOL;
	PLC_BA_DigIn_11 AT %QX0.15044.0:BOOL;
	PLC_BA_DigIn_12 AT %QX0.15048.0:BOOL;
	PLC_BA_DigIn_13 AT %QX0.15052.0:BOOL;
	PLC_BA_DigIn_14 AT %QX0.15056.0:BOOL;
	PLC_BA_DigIn_15 AT %QX0.15060.0:BOOL;
	PLC_BA_DigIn_16 AT %QX0.15064.0:BOOL;
	PLC_BA_DigIn_17 AT %QX0.15068.0:BOOL;
	PLC_BA_DigIn_18 AT %QX0.15072.0:BOOL;
	PLC_BA_DigIn_19 AT %QX0.15076.0:BOOL;
	PLC_BA_DigIn_20 AT %QX0.15080.0:BOOL;
	PLC_BA_DigIn_21 AT %QX0.15084.0:BOOL;
	PLC_BA_DigIn_22 AT %QX0.15088.0:BOOL;
	PLC_BA_DigIn_23 AT %QX0.15092.0:BOOL;
	PLC_BA_DigIn_24 AT %QX0.15096.0:BOOL;
	PLC_BA_DigIn_25 AT %QX0.15100.0:BOOL;
	PLC_BA_DigIn_26 AT %QX0.15104.0:BOOL;
	PLC_BA_DigIn_27 AT %QX0.15108.0:BOOL;
	PLC_BA_DigIn_28 AT %QX0.15112.0:BOOL;
	PLC_BA_DigIn_29 AT %QX0.15116.0:BOOL;
	PLC_BA_DigIn_30 AT %QX0.15120.0:BOOL;
	PLC_BA_DigIn_31 AT %QX0.15124.0:BOOL;
	PLC_BA_DigIn_32 AT %QX0.15128.0:BOOL;
	PLC_BA_OK_1 AT %QW0.15132:UINT;	(* 0=not visible 1=grey 2=yellow 3=green 4=red *)
	PLC_BA_OK_2 AT %QW0.15136:UINT;	(* 0=not visible 1=grey 2=yellow 3=green 4=red *)
	PLC_BA_OK_3 AT %QW0.15140:UINT;	(* 0=not visible 1=grey 2=yellow 3=green 4=red *)
	PLC_BA_OK_4 AT %QW0.15144:UINT;	(* 0=not visible 1=grey 2=yellow 3=green 4=red *)
	PLC_BA_OK_5 AT %QW0.15148:UINT;	(* 0=not visible 1=grey 2=yellow 3=green 4=red *)
	PLC_BA_OK_6 AT %QW0.15152:UINT;	(* 0=not visible 1=grey 2=yellow 3=green 4=red *)
	PLC_BA_OK_7 AT %QW0.15156:UINT;	(* 0=not visible 1=grey 2=yellow 3=green 4=red *)
	PLC_BA_OK_8 AT %QW0.15160:UINT;	(* 0=not visible 1=grey 2=yellow 3=green 4=red *)
	PLC_BA_OK_9 AT %QW0.15164:UINT;	(* 0=not visible 1=grey 2=yellow 3=green 4=red *)
	PLC_BA_OK_10 AT %QW0.15168:UINT;	(* 0=not visible 1=grey 2=yellow 3=green 4=red *)
	PLC_BA_OK_11 AT %QW0.15172:UINT;	(* 0=not visible 1=grey 2=yellow 3=green 4=red *)
	PLC_BA_OK_12 AT %QW0.15176:UINT;	(* 0=not visible 1=grey 2=yellow 3=green 4=red *)
	PLC_BA_OK_13 AT %QW0.15180:UINT;	(* 0=not visible 1=grey 2=yellow 3=green 4=red *)
	PLC_BA_OK_14 AT %QW0.15184:UINT;	(* 0=not visible 1=grey 2=yellow 3=green 4=red *)
	PLC_BA_OK_15 AT %QW0.15188:UINT;	(* 0=not visible 1=grey 2=yellow 3=green 4=red *)
	PLC_BA_OK_16 AT %QW0.15192:UINT;	(* 0=not visible 1=grey 2=yellow 3=green 4=red *)
	PLC_BA_OK_17 AT %QW0.15196:UINT;	(* 0=not visible 1=grey 2=yellow 3=green 4=red *)
	PLC_BA_OK_18 AT %QW0.15200:UINT;	(* 0=not visible 1=grey 2=yellow 3=green 4=red *)
	PLC_BA_OK_19 AT %QW0.15204:UINT;	(* 0=not visible 1=grey 2=yellow 3=green 4=red *)
	PLC_BA_OK_20 AT %QW0.15208:UINT;	(* 0=not visible 1=grey 2=yellow 3=green 4=red *)
	PLC_BA_OK_21 AT %QW0.15212:UINT;	(* 0=not visible 1=grey 2=yellow 3=green 4=red *)
	PLC_BA_OK_22 AT %QW0.15216:UINT;	(* 0=not visible 1=grey 2=yellow 3=green 4=red *)
	PLC_BA_OK_23 AT %QW0.15220:UINT;	(* 0=not visible 1=grey 2=yellow 3=green 4=red *)
	PLC_BA_OK_24 AT %QW0.15224:UINT;	(* 0=not visible 1=grey 2=yellow 3=green 4=red *)
	PLC_BA_OK_25 AT %QW0.15228:UINT;	(* 0=not visible 1=grey 2=yellow 3=green 4=red *)
	PLC_BA_OK_26 AT %QW0.15232:UINT;	(* 0=not visible 1=grey 2=yellow 3=green 4=red *)
	PLC_BA_OK_27 AT %QW0.15236:UINT;	(* 0=not visible 1=grey 2=yellow 3=green 4=red *)
	PLC_BA_OK_28 AT %QW0.15240:UINT;	(* 0=not visible 1=grey 2=yellow 3=green 4=red *)
	PLC_BA_OK_29 AT %QW0.15244:UINT;	(* 0=not visible 1=grey 2=yellow 3=green 4=red *)
	PLC_BA_OK_30 AT %QW0.15248:UINT;	(* 0=not visible 1=grey 2=yellow 3=green 4=red *)
	PLC_BA_OK_31 AT %QW0.15252:UINT;	(* 0=not visible 1=grey 2=yellow 3=green 4=red *)
	PLC_BA_OK_32 AT %QW0.15256:UINT;	(* 0=not visible 1=grey 2=yellow 3=green 4=red *)
	PLC_BA_control_type AT %QW0.15264:UINT;
	ARQ_FW AT %IW0.16000:UINT;	(* RTU0_STATUS NODE_10_STATUS *)
	ARQ_UPTIME_LED_h AT %ID0.16004:UDINT;
	ARQ_LIFETIME_RELE_h AT %ID0.16008:UDINT;
	ARQ_TCJ AT %IW0.16012:INT;
	ARQ_ERROR_ANOUT AT %IX0.16016.0:BOOL;
	ARQ_ERROR_STOUT AT %IX0.16020.0:BOOL;
	ARQ_ERROR_STOUT_A AT %IX0.16024.0:BOOL;
	ARQ_ERROR_WATCHDOG AT %IX0.16028.0:BOOL;
	ARQ_ERROR_SELFTEST_ON AT %IX0.16032.0:BOOL;
	ARQ_ERROR_PARAMETER AT %IX0.16036.0:BOOL;
	ARQ_ERROR_SELFTEST_DO1 AT %IX0.16040.0:BOOL;
	AQR_ERROR_SELFTEST_ANOUT AT %IX0.16044.0:BOOL;
	ARQ_AnOut AT %QW0.16048:INT;
	AQR_StOut AT %QW0.16052:UINT;
	ARQ_Rele AT %QX0.16056.0:BOOL;
	ARQ_reserved_1 AT %IW0.16060:UINT;
	ARQ_StOut_current AT %QW0.16064:INT;
	ARQ_Watchdog AT %QW0.16068:UINT;
	ARQ_Parity AT %QW0.16072:UINT;	(* 0=N 1=E 2=O *)
	ARQ_StopBits AT %QW0.16076:UINT;	(* 0=1bit 1=2bit *)
	ARQ_Baudrate AT %QW0.16080:UINT;	(* 0=9600 1=19200 2=38400 3=57600 *)
	ARQ_Address AT %QW0.16084:UINT;
	ARQ_PartNumber AT %QW0.16088:UINT;
	ARQ_reserved_2 AT %IW0.16092:UINT;
	ARQ_reserved_3 AT %IW0.16096:UINT;
	ARQ_reserved_4 AT %IW0.16100:UINT;
	ARQ_reserved_5 AT %IW0.16104:UINT;
	ARQ_SerialNumber AT %QW0.16108:UINT;
	ARQ_Setup AT %QW0.16112:UINT;	(* 0x5555 = save registers *)
	MPNE_A_FwRev AT %IW0.16116:UINT;	(* MPNE  firmware revision *)
	MPNE_A_ExpID AT %IW0.16120:UINT;	(* MPNE ID expansions *)
	MPNE_A_ExpType AT %IW0.16124:UINT;	(* MPNE  expansions type *)
	MPNE_A_SN AT %ID0.16128:UDINT;	(* MPNE serial number *)
	MPNE_A_LifeTime AT %ID0.16132:UDINT;	(* MPNE lifetime 1s *)
	MPNE_A_Status AT %IW0.16136:UINT;	(* MPNE status register *)
	MPNE_A_DigIn_1 AT %IX0.16140.0:BOOL;	(* Digital input 1 value *)
	MPNE_A_DigIn_2 AT %IX0.16144.0:BOOL;	(* Digital input 2 value *)
	MPNE_A_DigIn_3 AT %IX0.16148.0:BOOL;	(* Digital input 3 value *)
	MPNE_A_DigIn_4 AT %IX0.16152.0:BOOL;	(* Digital input 4 value *)
	MPNE_A_DigIn_5 AT %IX0.16156.0:BOOL;	(* Digital input 5 value *)
	MPNE_A_DigIn_6 AT %IX0.16160.0:BOOL;	(* Digital input 6 value *)
	MPNE_A_DigIn_7 AT %IX0.16164.0:BOOL;	(* Digital input 7 value *)
	MPNE_A_DigIn_8 AT %IX0.16168.0:BOOL;	(* Digital input 8 value *)
	MPNE_A_DigIn_9 AT %IX0.16172.0:BOOL;	(* Digital input 9 value *)
	MPNE_A_DigIn_10 AT %IX0.16176.0:BOOL;	(* Digital input 10 value *)
	MPNE_A_DigIn_11 AT %IX0.16180.0:BOOL;	(* Digital input 11 value *)
	MPNE_A_DigIn_12 AT %IX0.16184.0:BOOL;	(* Digital input 12 value *)
	MPNE_A_DigIn_13 AT %IX0.16188.0:BOOL;	(* Digital input 13 value *)
	MPNE_A_DigIn_14 AT %IX0.16192.0:BOOL;	(* Digital input 14 value *)
	MPNE_A_DigIn_15 AT %IX0.16196.0:BOOL;	(* Digital input 15 value *)
	MPNE_A_DigIn_16 AT %IX0.16200.0:BOOL;	(* Digital input 16 value *)
	MPNE_A_StatusWord AT %QW0.16304:UINT;	(* Fast Input Output Status Word *)
	MPNE_A_Watchdog AT %QW0.16308:UINT;	(* Watchdog *)
	MPNE_A_DigDir_1 AT %QX0.16312.0:BOOL;	(* Digital 1 direction (input = 0 output = 1) *)
	MPNE_A_DigDir_2 AT %QX0.16316.0:BOOL;	(* Digital 2 direction (input = 0 output = 1) *)
	MPNE_A_DigDir_3 AT %QX0.16320.0:BOOL;	(* Digital 3 direction (input = 0 output = 1) *)
	MPNE_A_DigDir_4 AT %QX0.16324.0:BOOL;	(* Digital 4 direction (input = 0 output = 1) *)
	MPNE_A_DigDir_5 AT %QX0.16328.0:BOOL;	(* Digital 5 direction (input = 0 output = 1) *)
	MPNE_A_DigDir_6 AT %QX0.16332.0:BOOL;	(* Digital 6 direction (input = 0 output = 1) *)
	MPNE_A_DigDir_7 AT %QX0.16336.0:BOOL;	(* Digital 7 direction (input = 0 output = 1) *)
	MPNE_A_DigDir_8 AT %QX0.16340.0:BOOL;	(* Digital 8 direction (input = 0 output = 1) *)
	MPNE_A_DigOut_1 AT %QX0.16344.0:BOOL;	(* Digital output 1 value *)
	MPNE_A_DigOut_2 AT %QX0.16348.0:BOOL;	(* Digital output 2 value *)
	MPNE_A_DigOut_3 AT %QX0.16352.0:BOOL;	(* Digital output 3 value *)
	MPNE_A_DigOut_4 AT %QX0.16356.0:BOOL;	(* Digital output 4 value *)
	MPNE_A_DigOut_5 AT %QX0.16360.0:BOOL;	(* Digital output 5 value *)
	MPNE_A_DigOut_6 AT %QX0.16364.0:BOOL;	(* Digital output 6 value *)
	MPNE_A_DigOut_7 AT %QX0.16368.0:BOOL;	(* Digital output 7 value *)
	MPNE_A_DigOut_8 AT %QX0.16372.0:BOOL;	(* Digital output 8 value *)
	MPNE_A_DigOut_17 AT %QX0.16376.0:BOOL;	(* Digital output 17 value *)
	MPNE_A_DigOut_18 AT %QX0.16380.0:BOOL;	(* Digital output 18 value *)
	MPNE_A_DigOut_19 AT %QX0.16384.0:BOOL;	(* Digital output 19 value *)
	MPNE_A_DigOut_20 AT %QX0.16388.0:BOOL;	(* Digital output 20 value *)
	MPNE_A_DigOut_21 AT %QX0.16392.0:BOOL;	(* Digital output 21 value *)
	MPNE_A_DigOut_22 AT %QX0.16396.0:BOOL;	(* Digital output 22 value *)
	MPNE_A_DigOut_23 AT %QX0.16400.0:BOOL;	(* Digital output 23 value *)
	MPNE_A_DigOut_24 AT %QX0.16404.0:BOOL;	(* Digital output 24 value *)
	MPNE_A_DigOut_25 AT %QX0.16408.0:BOOL;	(* Digital output 25 value *)
	MPNE_A_DigOut_26 AT %QX0.16412.0:BOOL;	(* Digital output 26 value *)
	MPNE_A_DigOut_27 AT %QX0.16416.0:BOOL;	(* Digital output 27 value *)
	MPNE_A_DigOut_28 AT %QX0.16420.0:BOOL;	(* Digital output 28 value *)
	MPNE_A_DigOut_29 AT %QX0.16424.0:BOOL;	(* Digital output 29 value *)
	MPNE_A_DigOut_30 AT %QX0.16428.0:BOOL;	(* Digital output 30 value *)
	MPNE_A_DigOut_31 AT %QX0.16432.0:BOOL;	(* Digital output 31 value *)
	MPNE_A_DigOut_32 AT %QX0.16436.0:BOOL;	(* Digital output 32 value *)
	MPNE_A_ControlWord_A AT %QW0.16440:UINT;	(* Fast Input Output Control Word  Line A *)
	MPNE_A_FastInDelay_A AT %QW0.16444:UINT;	(* Fast input delay time x 10us Line A *)
	MPNE_A_FastOutDelay_A AT %QW0.16448:UINT;	(* Fast output delay time x 10us Line A *)
	MPNE_A_FastOutDuration_A AT %QW0.16452:UINT;	(* Fast output duration time x 10us  Line A *)
	MPNE_A_EncCounter_A AT %QD0.16456:DINT;	(* Encoder Counter  Line A *)
	MPNE_A_MatchRegister_A AT %QD0.16460:DINT;	(* Match  Encoder  register  Line A *)
	MPNE_A_PTOTargetFreq_A AT %QW0.16464:UINT;	(* PTO Frequency Line A *)
	MPNE_A_PTOSteps_A AT %QD0.16468:UDINT;	(* PTO steps  Line A *)
	MPNE_B_FwRev AT %IW0.16648:UINT;	(* MPNE  firmware revision *)
	MPNE_B_ExpID AT %IW0.16652:UINT;	(* MPNE ID expansions *)
	MPNE_B_ExpType AT %IW0.16656:UINT;	(* MPNE  expansions type *)
	MPNE_B_SN AT %ID0.16660:UDINT;	(* MPNE serial number *)
	MPNE_B_LifeTime AT %ID0.16664:UDINT;	(* MPNE lifetime 1s *)
	MPNE_B_Status AT %IW0.16668:UINT;	(* MPNE status register *)
	MPNE_B_DigIn_1 AT %IX0.16672.0:BOOL;	(* Digital input 1 value *)
	MPNE_B_DigIn_2 AT %IX0.16676.0:BOOL;	(* Digital input 2 value *)
	MPNE_B_DigIn_3 AT %IX0.16680.0:BOOL;	(* Digital input 3 value *)
	MPNE_B_DigIn_4 AT %IX0.16684.0:BOOL;	(* Digital input 4 value *)
	MPNE_B_DigIn_5 AT %IX0.16688.0:BOOL;	(* Digital input 5 value *)
	MPNE_B_DigIn_6 AT %IX0.16692.0:BOOL;	(* Digital input 6 value *)
	MPNE_B_DigIn_7 AT %IX0.16696.0:BOOL;	(* Digital input 7 value *)
	MPNE_B_DigIn_8 AT %IX0.16700.0:BOOL;	(* Digital input 8 value *)
	MPNE_B_DigIn_9 AT %IX0.16704.0:BOOL;	(* Digital input 9 value *)
	MPNE_B_DigIn_10 AT %IX0.16708.0:BOOL;	(* Digital input 10 value *)
	MPNE_B_DigIn_11 AT %IX0.16712.0:BOOL;	(* Digital input 11 value *)
	MPNE_B_DigIn_12 AT %IX0.16716.0:BOOL;	(* Digital input 12 value *)
	MPNE_B_DigIn_13 AT %IX0.16720.0:BOOL;	(* Digital input 13 value *)
	MPNE_B_DigIn_14 AT %IX0.16724.0:BOOL;	(* Digital input 14 value *)
	MPNE_B_DigIn_15 AT %IX0.16728.0:BOOL;	(* Digital input 15 value *)
	MPNE_B_DigIn_16 AT %IX0.16732.0:BOOL;	(* Digital input 16 value *)
	MPNE_B_StatusWord AT %QW0.16836:UINT;	(* Fast Input Output Status Word *)
	MPNE_B_Watchdog AT %QW0.16840:UINT;	(* Watchdog *)
	MPNE_B_DigDir_1 AT %QX0.16844.0:BOOL;	(* Digital 1 direction (input = 0 output = 1) *)
	MPNE_B_DigDir_2 AT %QX0.16848.0:BOOL;	(* Digital 2 direction (input = 0 output = 1) *)
	MPNE_B_DigDir_3 AT %QX0.16852.0:BOOL;	(* Digital 3 direction (input = 0 output = 1) *)
	MPNE_B_DigDir_4 AT %QX0.16856.0:BOOL;	(* Digital 4 direction (input = 0 output = 1) *)
	MPNE_B_DigDir_5 AT %QX0.16860.0:BOOL;	(* Digital 5 direction (input = 0 output = 1) *)
	MPNE_B_DigDir_6 AT %QX0.16864.0:BOOL;	(* Digital 6 direction (input = 0 output = 1) *)
	MPNE_B_DigDir_7 AT %QX0.16868.0:BOOL;	(* Digital 7 direction (input = 0 output = 1) *)
	MPNE_B_DigDir_8 AT %QX0.16872.0:BOOL;	(* Digital 8 direction (input = 0 output = 1) *)
	MPNE_B_DigOut_1 AT %QX0.16876.0:BOOL;	(* Digital output 1 value *)
	MPNE_B_DigOut_2 AT %QX0.16880.0:BOOL;	(* Digital output 2 value *)
	MPNE_B_DigOut_3 AT %QX0.16884.0:BOOL;	(* Digital output 3 value *)
	MPNE_B_DigOut_4 AT %QX0.16888.0:BOOL;	(* Digital output 4 value *)
	MPNE_B_DigOut_5 AT %QX0.16892.0:BOOL;	(* Digital output 5 value *)
	MPNE_B_DigOut_6 AT %QX0.16896.0:BOOL;	(* Digital output 6 value *)
	MPNE_B_DigOut_7 AT %QX0.16900.0:BOOL;	(* Digital output 7 value *)
	MPNE_B_DigOut_8 AT %QX0.16904.0:BOOL;	(* Digital output 8 value *)
	MPNE_B_DigOut_17 AT %QX0.16908.0:BOOL;	(* Digital output 17 value *)
	MPNE_B_DigOut_18 AT %QX0.16912.0:BOOL;	(* Digital output 18 value *)
	MPNE_B_DigOut_19 AT %QX0.16916.0:BOOL;	(* Digital output 19 value *)
	MPNE_B_DigOut_20 AT %QX0.16920.0:BOOL;	(* Digital output 20 value *)
	MPNE_B_DigOut_21 AT %QX0.16924.0:BOOL;	(* Digital output 21 value *)
	MPNE_B_DigOut_22 AT %QX0.16928.0:BOOL;	(* Digital output 22 value *)
	MPNE_B_DigOut_23 AT %QX0.16932.0:BOOL;	(* Digital output 23 value *)
	MPNE_B_DigOut_24 AT %QX0.16936.0:BOOL;	(* Digital output 24 value *)
	MPNE_B_DigOut_25 AT %QX0.16940.0:BOOL;	(* Digital output 25 value *)
	MPNE_B_DigOut_26 AT %QX0.16944.0:BOOL;	(* Digital output 26 value *)
	MPNE_B_DigOut_27 AT %QX0.16948.0:BOOL;	(* Digital output 27 value *)
	MPNE_B_DigOut_28 AT %QX0.16952.0:BOOL;	(* Digital output 28 value *)
	MPNE_B_DigOut_29 AT %QX0.16956.0:BOOL;	(* Digital output 29 value *)
	MPNE_B_DigOut_30 AT %QX0.16960.0:BOOL;	(* Digital output 30 value *)
	MPNE_B_DigOut_31 AT %QX0.16964.0:BOOL;	(* Digital output 31 value *)
	MPNE_B_DigOut_32 AT %QX0.16968.0:BOOL;	(* Digital output 32 value *)
	MPNE_B_ControlWord_A AT %QW0.16972:UINT;	(* Fast Input Output Control Word  Line A *)
	MPNE_B_FastInDelay_A AT %QW0.16976:UINT;	(* Fast input delay time x 10us Line A *)
	MPNE_B_FastOutDelay_A AT %QW0.16980:UINT;	(* Fast output delay time x 10us Line A *)
	MPNE_B_FastOutDuration_A AT %QW0.16984:UINT;	(* Fast output duration time x 10us  Line A *)
	MPNE_B_EncCounter_A AT %QD0.16988:DINT;	(* Encoder Counter  Line A *)
	MPNE_B_MatchRegister_A AT %QD0.16992:DINT;	(* Match  Encoder  register  Line A *)
	MPNE_B_PTOTargetFreq_A AT %QW0.16996:UINT;	(* PTO Frequency Line A *)
	MPNE_B_PTOSteps_A AT %QD0.17000:UDINT;	(* PTO steps  Line A *)
	MPNE_C_FwRev AT %IW0.17180:UINT;	(* MPNE  firmware revision *)
	MPNE_C_ExpID AT %IW0.17184:UINT;	(* MPNE ID expansions *)
	MPNE_C_ExpType AT %IW0.17188:UINT;	(* MPNE  expansions type *)
	MPNE_C_SN AT %ID0.17192:UDINT;	(* MPNE serial number *)
	MPNE_C_LifeTime AT %ID0.17196:UDINT;	(* MPNE lifetime 1s *)
	MPNE_C_Status AT %IW0.17200:UINT;	(* MPNE status register *)
	MPNE_C_DigIn_1 AT %IX0.17204.0:BOOL;	(* Digital input 1 value *)
	MPNE_C_DigIn_2 AT %IX0.17208.0:BOOL;	(* Digital input 2 value *)
	MPNE_C_DigIn_3 AT %IX0.17212.0:BOOL;	(* Digital input 3 value *)
	MPNE_C_DigIn_4 AT %IX0.17216.0:BOOL;	(* Digital input 4 value *)
	MPNE_C_DigIn_5 AT %IX0.17220.0:BOOL;	(* Digital input 5 value *)
	MPNE_C_DigIn_6 AT %IX0.17224.0:BOOL;	(* Digital input 6 value *)
	MPNE_C_DigIn_7 AT %IX0.17228.0:BOOL;	(* Digital input 7 value *)
	MPNE_C_DigIn_8 AT %IX0.17232.0:BOOL;	(* Digital input 8 value *)
	MPNE_C_DigIn_9 AT %IX0.17236.0:BOOL;	(* Digital input 9 value *)
	MPNE_C_DigIn_10 AT %IX0.17240.0:BOOL;	(* Digital input 10 value *)
	MPNE_C_DigIn_11 AT %IX0.17244.0:BOOL;	(* Digital input 11 value *)
	MPNE_C_DigIn_12 AT %IX0.17248.0:BOOL;	(* Digital input 12 value *)
	MPNE_C_DigIn_13 AT %IX0.17252.0:BOOL;	(* Digital input 13 value *)
	MPNE_C_DigIn_14 AT %IX0.17256.0:BOOL;	(* Digital input 14 value *)
	MPNE_C_DigIn_15 AT %IX0.17260.0:BOOL;	(* Digital input 15 value *)
	MPNE_C_DigIn_16 AT %IX0.17264.0:BOOL;	(* Digital input 16 value *)
	MPNE_C_AnIn_1 AT %IW0.17332:INT;	(* Analog input 1 value *)
	MPNE_C_AnIn_2 AT %IW0.17336:INT;	(* Analog input 2 value *)
	MPNE_C_AnIn_3 AT %IW0.17340:INT;	(* Analog input 3 value *)
	MPNE_C_AnIn_4 AT %IW0.17344:INT;	(* Analog input 4 value *)
	MPNE_C_AnInStatus AT %IW0.17348:INT;	(* Analog Inputs status register *)
	MPNE_C_StatusWord AT %QW0.17368:UINT;	(* Fast Input Output Status Word *)
	MPNE_C_Watchdog AT %QW0.17372:UINT;	(* Watchdog *)
	MPNE_C_DigDir_1 AT %QX0.17376.0:BOOL;	(* Digital 1 direction (input = 0 output = 1) *)
	MPNE_C_DigDir_2 AT %QX0.17380.0:BOOL;	(* Digital 2 direction (input = 0 output = 1) *)
	MPNE_C_DigDir_3 AT %QX0.17384.0:BOOL;	(* Digital 3 direction (input = 0 output = 1) *)
	MPNE_C_DigDir_4 AT %QX0.17388.0:BOOL;	(* Digital 4 direction (input = 0 output = 1) *)
	MPNE_C_DigDir_5 AT %QX0.17392.0:BOOL;	(* Digital 5 direction (input = 0 output = 1) *)
	MPNE_C_DigDir_6 AT %QX0.17396.0:BOOL;	(* Digital 6 direction (input = 0 output = 1) *)
	MPNE_C_DigDir_7 AT %QX0.17400.0:BOOL;	(* Digital 7 direction (input = 0 output = 1) *)
	MPNE_C_DigDir_8 AT %QX0.17404.0:BOOL;	(* Digital 8 direction (input = 0 output = 1) *)
	MPNE_C_DigOut_1 AT %QX0.17408.0:BOOL;	(* Digital output 1 value *)
	MPNE_C_DigOut_2 AT %QX0.17412.0:BOOL;	(* Digital output 2 value *)
	MPNE_C_DigOut_3 AT %QX0.17416.0:BOOL;	(* Digital output 3 value *)
	MPNE_C_DigOut_4 AT %QX0.17420.0:BOOL;	(* Digital output 4 value *)
	MPNE_C_DigOut_5 AT %QX0.17424.0:BOOL;	(* Digital output 5 value *)
	MPNE_C_DigOut_6 AT %QX0.17428.0:BOOL;	(* Digital output 6 value *)
	MPNE_C_DigOut_7 AT %QX0.17432.0:BOOL;	(* Digital output 7 value *)
	MPNE_C_DigOut_8 AT %QX0.17436.0:BOOL;	(* Digital output 8 value *)
	MPNE_C_ControlWord_A AT %QW0.17504:UINT;	(* Fast Input Output Control Word  Line A *)
	MPNE_C_FastInDelay_A AT %QW0.17508:UINT;	(* Fast input delay time x 10us Line A *)
	MPNE_C_FastOutDelay_A AT %QW0.17512:UINT;	(* Fast output delay time x 10us Line A *)
	MPNE_C_FastOutDuration_A AT %QW0.17516:UINT;	(* Fast output duration time x 10us  Line A *)
	MPNE_C_EncCounter_A AT %QD0.17520:DINT;	(* Encoder Counter  Line A *)
	MPNE_C_MatchRegister_A AT %QD0.17524:DINT;	(* Match  Encoder  register  Line A *)
	MPNE_C_PTOTargetFreq_A AT %QW0.17528:UINT;	(* PTO Frequency Line A *)
	MPNE_C_PTOSteps_A AT %QD0.17532:UDINT;	(* PTO steps  Line A *)
	MPNE_C_AnIn1Conf AT %QW0.17664:UINT;	(* Analog input 1 configuration *)
	MPNE_C_AnIn2Conf AT %QW0.17668:UINT;	(* Analog input 2 configuration *)
	MPNE_C_AnIn3Conf AT %QW0.17672:UINT;	(* Analog input 3 configuration *)
	MPNE_C_AnIn4Conf AT %QW0.17676:UINT;	(* Analog input 4 configuration *)
	MPNE_C_AnOut1Conf AT %QW0.17680:UINT;	(* Analog output 1 configuration *)
	MPNE_C_AnOut2Conf AT %QW0.17684:UINT;	(* Analog output 2 configuration *)
	MPNE_C_AnOut1 AT %QW0.17688:UINT;	(* Analog output 1 value *)
	MPNE_C_AnOut2 AT %QW0.17692:UINT;	(* Analog output 2 value *)
	MPNE_C_AnIn1Filter AT %QW0.17696:UINT;	(* Analog input 1 filter *)
	MPNE_C_AnIn2Filter AT %QW0.17700:UINT;	(* Analog input 2 filter *)
	MPNE_C_AnIn3Filter AT %QW0.17704:UINT;	(* Analog input 3 filter *)
	MPNE_C_AnIn4Filter AT %QW0.17708:UINT;	(* Analog input 4 filter *)
	MPNE_D_FwRev AT %IW0.17712:UINT;	(* MPNE  firmware revision *)
	MPNE_D_ExpID AT %IW0.17716:UINT;	(* MPNE ID expansions *)
	MPNE_D_ExpType AT %IW0.17720:UINT;	(* MPNE  expansions type *)
	MPNE_D_SN AT %ID0.17724:UDINT;	(* MPNE serial number *)
	MPNE_D_LifeTime AT %ID0.17728:UDINT;	(* MPNE lifetime 1s *)
	MPNE_D_Status AT %IW0.17732:UINT;	(* MPNE status register *)
	MPNE_D_DigIn_1 AT %IX0.17736.0:BOOL;	(* Digital input 1 value *)
	MPNE_D_DigIn_2 AT %IX0.17740.0:BOOL;	(* Digital input 2 value *)
	MPNE_D_DigIn_3 AT %IX0.17744.0:BOOL;	(* Digital input 3 value *)
	MPNE_D_DigIn_4 AT %IX0.17748.0:BOOL;	(* Digital input 4 value *)
	MPNE_D_DigIn_5 AT %IX0.17752.0:BOOL;	(* Digital input 5 value *)
	MPNE_D_DigIn_6 AT %IX0.17756.0:BOOL;	(* Digital input 6 value *)
	MPNE_D_DigIn_7 AT %IX0.17760.0:BOOL;	(* Digital input 7 value *)
	MPNE_D_DigIn_8 AT %IX0.17764.0:BOOL;	(* Digital input 8 value *)
	MPNE_D_DigIn_9 AT %IX0.17768.0:BOOL;	(* Digital input 9 value *)
	MPNE_D_DigIn_10 AT %IX0.17772.0:BOOL;	(* Digital input 10 value *)
	MPNE_D_DigIn_11 AT %IX0.17776.0:BOOL;	(* Digital input 11 value *)
	MPNE_D_DigIn_12 AT %IX0.17780.0:BOOL;	(* Digital input 12 value *)
	MPNE_D_DigIn_13 AT %IX0.17784.0:BOOL;	(* Digital input 13 value *)
	MPNE_D_DigIn_14 AT %IX0.17788.0:BOOL;	(* Digital input 14 value *)
	MPNE_D_DigIn_15 AT %IX0.17792.0:BOOL;	(* Digital input 15 value *)
	MPNE_D_DigIn_16 AT %IX0.17796.0:BOOL;	(* Digital input 16 value *)
	MPNE_D_AnIn_1 AT %IW0.17864:INT;	(* Analog input 1 value *)
	MPNE_D_AnIn_2 AT %IW0.17868:INT;	(* Analog input 2 value *)
	MPNE_D_AnIn_3 AT %IW0.17872:INT;	(* Analog input 3 value *)
	MPNE_D_AnIn_4 AT %IW0.17876:INT;	(* Analog input 4 value *)
	MPNE_D_AnInStatus AT %IW0.17880:INT;	(* Analog Inputs status register *)
	MPNE_D_StatusWord AT %QW0.17900:UINT;	(* Fast Input Output Status Word *)
	MPNE_D_Watchdog AT %QW0.17904:UINT;	(* Watchdog *)
	MPNE_D_DigDir_1 AT %QX0.17908.0:BOOL;	(* Digital 1 direction (input = 0 output = 1) *)
	MPNE_D_DigDir_2 AT %QX0.17912.0:BOOL;	(* Digital 2 direction (input = 0 output = 1) *)
	MPNE_D_DigDir_3 AT %QX0.17916.0:BOOL;	(* Digital 3 direction (input = 0 output = 1) *)
	MPNE_D_DigDir_4 AT %QX0.17920.0:BOOL;	(* Digital 4 direction (input = 0 output = 1) *)
	MPNE_D_DigDir_5 AT %QX0.17924.0:BOOL;	(* Digital 5 direction (input = 0 output = 1) *)
	MPNE_D_DigDir_6 AT %QX0.17928.0:BOOL;	(* Digital 6 direction (input = 0 output = 1) *)
	MPNE_D_DigDir_7 AT %QX0.17932.0:BOOL;	(* Digital 7 direction (input = 0 output = 1) *)
	MPNE_D_DigDir_8 AT %QX0.17936.0:BOOL;	(* Digital 8 direction (input = 0 output = 1) *)
	MPNE_D_DigOut_1 AT %QX0.17940.0:BOOL;	(* Digital output 1 value *)
	MPNE_D_DigOut_2 AT %QX0.17944.0:BOOL;	(* Digital output 2 value *)
	MPNE_D_DigOut_3 AT %QX0.17948.0:BOOL;	(* Digital output 3 value *)
	MPNE_D_DigOut_4 AT %QX0.17952.0:BOOL;	(* Digital output 4 value *)
	MPNE_D_DigOut_5 AT %QX0.17956.0:BOOL;	(* Digital output 5 value *)
	MPNE_D_DigOut_6 AT %QX0.17960.0:BOOL;	(* Digital output 6 value *)
	MPNE_D_DigOut_7 AT %QX0.17964.0:BOOL;	(* Digital output 7 value *)
	MPNE_D_DigOut_8 AT %QX0.17968.0:BOOL;	(* Digital output 8 value *)
	MPNE_D_ControlWord_A AT %QW0.18036:UINT;	(* Fast Input Output Control Word  Line A *)
	MPNE_D_FastInDelay_A AT %QW0.18040:UINT;	(* Fast input delay time x 10us Line A *)
	MPNE_D_FastOutDelay_A AT %QW0.18044:UINT;	(* Fast output delay time x 10us Line A *)
	MPNE_D_FastOutDuration_A AT %QW0.18048:UINT;	(* Fast output duration time x 10us  Line A *)
	MPNE_D_EncCounter_A AT %QD0.18052:DINT;	(* Encoder Counter  Line A *)
	MPNE_D_MatchRegister_A AT %QD0.18056:DINT;	(* Match  Encoder  register  Line A *)
	MPNE_D_PTOTargetFreq_A AT %QW0.18060:UINT;	(* PTO Frequency Line A *)
	MPNE_D_PTOSteps_A AT %QD0.18064:UDINT;	(* PTO steps  Line A *)
	MPNE_D_AnIn1Conf AT %QW0.18196:UINT;	(* Analog input 1 configuration *)
	MPNE_D_AnIn2Conf AT %QW0.18200:UINT;	(* Analog input 2 configuration *)
	MPNE_D_AnIn3Conf AT %QW0.18204:UINT;	(* Analog input 3 configuration *)
	MPNE_D_AnIn4Conf AT %QW0.18208:UINT;	(* Analog input 4 configuration *)
	MPNE_D_AnOut1Conf AT %QW0.18212:UINT;	(* Analog output 1 configuration *)
	MPNE_D_AnOut2Conf AT %QW0.18216:UINT;	(* Analog output 2 configuration *)
	MPNE_D_AnOut1 AT %QW0.18220:UINT;	(* Analog output 1 value *)
	MPNE_D_AnOut2 AT %QW0.18224:UINT;	(* Analog output 2 value *)
	MPNE_D_AnIn1Filter AT %QW0.18228:UINT;	(* Analog input 1 filter *)
	MPNE_D_AnIn2Filter AT %QW0.18232:UINT;	(* Analog input 2 filter *)
	MPNE_D_AnIn3Filter AT %QW0.18236:UINT;	(* Analog input 3 filter *)
	MPNE_D_AnIn4Filter AT %QW0.18240:UINT;	(* Analog input 4 filter *)
	RTU_EP_wattmeter_M_P AT %ID0.18244:REAL;	(* active power +/- xxxx.xxx W *)
	RTU_EP_wattmeter_M_Q AT %ID0.18248:REAL;	(* reactive power +/- xxxx.xxx var *)
	RTU_EP_wattmeter_M_S AT %ID0.18252:REAL;	(* apparent power +/- xxxx.xxx VA *)
	RTU_EP_wattmeter_M_C AT %ID0.18256:REAL;	(* power factor +/- x.xxx *)
	RTU_EP_wattmeter_M_F AT %ID0.18260:REAL;	(* frequency xx.xxx Hz *)
	RTU_EP_wattmeter_M_U AT %ID0.18264:REAL;	(* voltage xxx.xx V *)
	RTU_EP_wattmeter_M_I1 AT %ID0.18268:REAL;	(* current xx.xxx A (1) *)
	RTU_EP_wattmeter_M_I2 AT %ID0.18272:REAL;	(* current xx.xxx A (2) *)
	RTU_EP_wattmeter_M_I3 AT %ID0.18276:REAL;	(* current xx.xxx A (3) *)
	RTU_EP_wattmeter_M_I AT %ID0.18280:REAL;	(* current xx.xxx A *)
	RTU_EP_wattmeter_M_Ein AT %ID0.18284:REAL;	(* imported energy xxxxxxxxx.x Wh *)
	RTU_EP_wattmeter_M_Eout AT %ID0.18288:REAL;	(* exported energy xxxxxxxxx.x Wh *)
	RTU_EP_wattmeter_F_P AT %ID0.18292:REAL;	(* active power +/- xxxx.xxx W *)
	RTU_EP_wattmeter_F_Q AT %ID0.18296:REAL;	(* reactive power +/- xxxx.xxx var *)
	RTU_EP_wattmeter_F_S AT %ID0.18300:REAL;	(* apparent power +/- xxxx.xxx VA *)
	RTU_EP_wattmeter_F_C AT %ID0.18304:REAL;	(* power factor +/- x.xxx *)
	RTU_EP_wattmeter_F_F AT %ID0.18308:REAL;	(* frequency xx.xxx Hz *)
	RTU_EP_wattmeter_F_U AT %ID0.18312:REAL;	(* voltage xxx.xx V *)
	RTU_EP_wattmeter_F_I1 AT %ID0.18316:REAL;	(* current xx.xxx A (1) *)
	RTU_EP_wattmeter_F_I2 AT %ID0.18320:REAL;	(* current xx.xxx A (2) *)
	RTU_EP_wattmeter_F_I3 AT %ID0.18324:REAL;	(* current xx.xxx A (3) *)
	RTU_EP_wattmeter_F_I AT %ID0.18328:REAL;	(* current xx.xxx A *)
	RTU_EP_wattmeter_F_Ein AT %ID0.18332:REAL;	(* imported energy xxxxxxxxx.x Wh *)
	RTU_EP_wattmeter_F_Eout AT %ID0.18336:REAL;	(* exported energy xxxxxxxxx.x Wh *)
	RTU_EP_wattmeter01_P AT %ID0.18340:REAL;	(* active power +/- xxxx.xxx W *)
	RTU_EP_wattmeter01_Q AT %ID0.18344:REAL;	(* reactive power +/- xxxx.xxx var *)
	RTU_EP_wattmeter01_S AT %ID0.18348:REAL;	(* apparent power +/- xxxx.xxx VA *)
	RTU_EP_wattmeter01_Ein AT %ID0.18352:REAL;	(* imported energy xxxxxxxxx.x Wh *)
	RTU_EP_wattmeter02_P AT %ID0.18356:REAL;	(* active power +/- xxxx.xxx W *)
	RTU_EP_wattmeter02_Q AT %ID0.18360:REAL;	(* reactive power +/- xxxx.xxx var *)
	RTU_EP_wattmeter02_S AT %ID0.18364:REAL;	(* apparent power +/- xxxx.xxx VA *)
	RTU_EP_wattmeter02_Ein AT %ID0.18368:REAL;	(* imported energy xxxxxxxxx.x Wh *)
	RTU_EP_wattmeter03_P AT %ID0.18372:REAL;	(* active power +/- xxxx.xxx W *)
	RTU_EP_wattmeter03_Q AT %ID0.18376:REAL;	(* reactive power +/- xxxx.xxx var *)
	RTU_EP_wattmeter03_S AT %ID0.18380:REAL;	(* apparent power +/- xxxx.xxx VA *)
	RTU_EP_wattmeter03_Ein AT %ID0.18384:REAL;	(* imported energy xxxxxxxxx.x Wh *)
	RTU_EP_wattmeter04_P AT %ID0.18388:REAL;	(* active power +/- xxxx.xxx W *)
	RTU_EP_wattmeter04_Q AT %ID0.18392:REAL;	(* reactive power +/- xxxx.xxx var *)
	RTU_EP_wattmeter04_S AT %ID0.18396:REAL;	(* apparent power +/- xxxx.xxx VA *)
	RTU_EP_wattmeter04_Ein AT %ID0.18400:REAL;	(* imported energy xxxxxxxxx.x Wh *)
	RTU_EP_wattmeter05_P AT %ID0.18404:REAL;	(* active power +/- xxxx.xxx W *)
	RTU_EP_wattmeter05_Q AT %ID0.18408:REAL;	(* reactive power +/- xxxx.xxx var *)
	RTU_EP_wattmeter05_S AT %ID0.18412:REAL;	(* apparent power +/- xxxx.xxx VA *)
	RTU_EP_wattmeter05_Ein AT %ID0.18416:REAL;	(* imported energy xxxxxxxxx.x Wh *)
	RTU_EP_wattmeter06_P AT %ID0.18420:REAL;	(* active power +/- xxxx.xxx W *)
	RTU_EP_wattmeter06_Q AT %ID0.18424:REAL;	(* reactive power +/- xxxx.xxx var *)
	RTU_EP_wattmeter06_S AT %ID0.18428:REAL;	(* apparent power +/- xxxx.xxx VA *)
	RTU_EP_wattmeter06_Ein AT %ID0.18432:REAL;	(* imported energy xxxxxxxxx.x Wh *)
	RTU_EP_wattmeter07_P AT %ID0.18436:REAL;	(* active power +/- xxxx.xxx W *)
	RTU_EP_wattmeter07_Q AT %ID0.18440:REAL;	(* reactive power +/- xxxx.xxx var *)
	RTU_EP_wattmeter07_S AT %ID0.18444:REAL;	(* apparent power +/- xxxx.xxx VA *)
	RTU_EP_wattmeter07_Ein AT %ID0.18448:REAL;	(* imported energy xxxxxxxxx.x Wh *)
	RTU_EP_wattmeter08_P AT %ID0.18452:REAL;	(* active power +/- xxxx.xxx W *)
	RTU_EP_wattmeter08_Q AT %ID0.18456:REAL;	(* reactive power +/- xxxx.xxx var *)
	RTU_EP_wattmeter08_S AT %ID0.18460:REAL;	(* apparent power +/- xxxx.xxx VA *)
	RTU_EP_wattmeter08_Ein AT %ID0.18464:REAL;	(* imported energy xxxxxxxxx.x Wh *)
	RTU_EP_wattmeter09_P AT %ID0.18468:REAL;	(* active power +/- xxxx.xxx W *)
	RTU_EP_wattmeter09_Q AT %ID0.18472:REAL;	(* reactive power +/- xxxx.xxx var *)
	RTU_EP_wattmeter09_S AT %ID0.18476:REAL;	(* apparent power +/- xxxx.xxx VA *)
	RTU_EP_wattmeter09_Ein AT %ID0.18480:REAL;	(* imported energy xxxxxxxxx.x Wh *)
	RTU_EP_wattmeter10_P AT %ID0.18484:REAL;	(* active power +/- xxxx.xxx W *)
	RTU_EP_wattmeter10_Q AT %ID0.18488:REAL;	(* reactive power +/- xxxx.xxx var *)
	RTU_EP_wattmeter10_S AT %ID0.18492:REAL;	(* apparent power +/- xxxx.xxx VA *)
	RTU_EP_wattmeter10_Ein AT %ID0.18496:REAL;	(* imported energy xxxxxxxxx.x Wh *)
	MPNC_Baudrate AT %IW0.18500:UINT;	(* Baudrate MPNC006 device *)
	MPNC_NodeID AT %IW0.18504:UINT;	(* Address MPNC006 device *)
	MPNC_HeartBeat AT %ID0.18508:UDINT;	(* Life time MPNC006 device *)
	MPNC_AnInConf_A AT %QW0.18512:UINT;	(* Analog inputs configuration MPNC030 module A *)
	MPNC_AnInConf_B AT %QW0.18516:UINT;	(* Analog inputs configuration MPNC030 module B *)
	MPNC_AnInConf_C AT %QW0.18520:UINT;	(* Analog inputs configuration MPNC030 module C *)
	MPNC_AnInConf_D AT %QW0.18524:UINT;	(* Analog inputs configuration MPNC030 module D *)
	MPNC_AnIn_A_1 AT %IW0.18528:INT;	(* Analog input 1 value MPNC030 module A *)
	MPNC_AnIn_A_2 AT %IW0.18532:INT;	(* Analog input 2 value MPNC030 module A *)
	MPNC_AnIn_A_3 AT %IW0.18536:INT;	(* Analog input 3 value MPNC030 module A *)
	MPNC_AnIn_A_4 AT %IW0.18540:INT;	(* Analog input 4 value MPNC030 module A *)
	MPNC_AnIn_B_1 AT %IW0.18544:INT;	(* Analog input 1 value MPNC030 module B *)
	MPNC_AnIn_B_2 AT %IW0.18548:INT;	(* Analog input 2 value MPNC030 module B *)
	MPNC_AnIn_B_3 AT %IW0.18552:INT;	(* Analog input 3 value MPNC030 module B *)
	MPNC_AnIn_B_4 AT %IW0.18556:INT;	(* Analog input 4 value MPNC030 module B *)
	MPNC_AnIn_C_1 AT %IW0.18560:INT;	(* Analog input 1 value MPNC030 module C *)
	MPNC_AnIn_C_2 AT %IW0.18564:INT;	(* Analog input 2 value MPNC030 module C *)
	MPNC_AnIn_C_3 AT %IW0.18568:INT;	(* Analog input 3 value MPNC030 module C *)
	MPNC_AnIn_C_4 AT %IW0.18572:INT;	(* Analog input 4 value MPNC030 module C *)
	MPNC_AnIn_D_1 AT %IW0.18576:INT;	(* Analog input 1 value MPNC030 module D *)
	MPNC_AnIn_D_2 AT %IW0.18580:INT;	(* Analog input 2 value MPNC030 module D *)
	MPNC_AnIn_D_3 AT %IW0.18584:INT;	(* Analog input 3 value MPNC030 module D *)
	MPNC_AnIn_D_4 AT %IW0.18588:INT;	(* Analog input 4 value MPNC030 module D *)
	MPNC_DigOut_A_1 AT %QX0.18592.0:BOOL;	(* Digital output value bit 1 MPNC020 02 module A *)
	MPNC_DigOut_A_2 AT %QX0.18596.0:BOOL;	(* Digital output value bit 2 MPNC020 02 module A *)
	MPNC_DigOut_A_3 AT %QX0.18600.0:BOOL;	(* Digital output value bit 3 MPNC020 02 module A *)
	MPNC_DigOut_A_4 AT %QX0.18604.0:BOOL;	(* Digital output value bit 4 MPNC020 02 module A *)
	MPNC_DigOut_A_5 AT %QX0.18608.0:BOOL;	(* Digital output value bit 5 MPNC020 02 module A *)
	MPNC_DigOut_A_6 AT %QX0.18612.0:BOOL;	(* Digital output value bit 6 MPNC020 02 module A *)
	MPNC_DigOut_A_7 AT %QX0.18616.0:BOOL;	(* Digital output value bit 7 MPNC020 02 module A *)
	MPNC_DigOut_A_8 AT %QX0.18620.0:BOOL;	(* Digital output value bit 8 MPNC020 02 module A *)
	MPNC_DigOut_A_9 AT %QX0.18624.0:BOOL;	(* Digital output value bit 9 MPNC020 02 module A *)
	MPNC_DigOut_A_10 AT %QX0.18628.0:BOOL;	(* Digital output value bit 10 MPNC020 02 module A *)
	MPNC_DigOut_A_11 AT %QX0.18632.0:BOOL;	(* Digital output value bit 11 MPNC020 02 module A *)
	MPNC_DigOut_A_12 AT %QX0.18636.0:BOOL;	(* Digital output value bit 12 MPNC020 02 module A *)
	MPNC_DigOut_A_13 AT %QX0.18640.0:BOOL;	(* Digital output value bit 13 MPNC020 02 module A *)
	MPNC_DigOut_A_14 AT %QX0.18644.0:BOOL;	(* Digital output value bit 14 MPNC020 02 module A *)
	MPNC_DigOut_A_15 AT %QX0.18648.0:BOOL;	(* Digital output value bit 15 MPNC020 02 module A *)
	MPNC_DigOut_A_16 AT %QX0.18652.0:BOOL;	(* Digital output value bit 16 MPNC020 02 module A *)
	MPNC_DigOut_B_1 AT %QX0.18656.0:BOOL;	(* Digital output value bit 1 MPNC020 02 module B *)
	MPNC_DigOut_B_2 AT %QX0.18660.0:BOOL;	(* Digital output value bit 2 MPNC020 02 module B *)
	MPNC_DigOut_B_3 AT %QX0.18664.0:BOOL;	(* Digital output value bit 3 MPNC020 02 module B *)
	MPNC_DigOut_B_4 AT %QX0.18668.0:BOOL;	(* Digital output value bit 4 MPNC020 02 module B *)
	MPNC_DigOut_B_5 AT %QX0.18672.0:BOOL;	(* Digital output value bit 5 MPNC020 02 module B *)
	MPNC_DigOut_B_6 AT %QX0.18676.0:BOOL;	(* Digital output value bit 6 MPNC020 02 module B *)
	MPNC_DigOut_B_7 AT %QX0.18680.0:BOOL;	(* Digital output value bit 7 MPNC020 02 module B *)
	MPNC_DigOut_B_8 AT %QX0.18684.0:BOOL;	(* Digital output value bit 8 MPNC020 02 module B *)
	MPNC_DigOut_B_9 AT %QX0.18688.0:BOOL;	(* Digital output value bit 9 MPNC020 02 module B *)
	MPNC_DigOut_B_10 AT %QX0.18692.0:BOOL;	(* Digital output value bit 10 MPNC020 02 module B *)
	MPNC_DigOut_B_11 AT %QX0.18696.0:BOOL;	(* Digital output value bit 11 MPNC020 02 module B *)
	MPNC_DigOut_B_12 AT %QX0.18700.0:BOOL;	(* Digital output value bit 12 MPNC020 02 module B *)
	MPNC_DigOut_B_13 AT %QX0.18704.0:BOOL;	(* Digital output value bit 13 MPNC020 02 module B *)
	MPNC_DigOut_B_14 AT %QX0.18708.0:BOOL;	(* Digital output value bit 14 MPNC020 02 module B *)
	MPNC_DigOut_B_15 AT %QX0.18712.0:BOOL;	(* Digital output value bit 15 MPNC020 02 module B *)
	MPNC_DigOut_B_16 AT %QX0.18716.0:BOOL;	(* Digital output value bit 16 MPNC020 02 module B *)
	MPNC_DigOut_C_1 AT %QX0.18720.0:BOOL;	(* Digital output value bit 1 MPNC020 02 module C *)
	MPNC_DigOut_C_2 AT %QX0.18724.0:BOOL;	(* Digital output value bit 2 MPNC020 02 module C *)
	MPNC_DigOut_C_3 AT %QX0.18728.0:BOOL;	(* Digital output value bit 3 MPNC020 02 module C *)
	MPNC_DigOut_C_4 AT %QX0.18732.0:BOOL;	(* Digital output value bit 4 MPNC020 02 module C *)
	MPNC_DigOut_C_5 AT %QX0.18736.0:BOOL;	(* Digital output value bit 5 MPNC020 02 module C *)
	MPNC_DigOut_C_6 AT %QX0.18740.0:BOOL;	(* Digital output value bit 6 MPNC020 02 module C *)
	MPNC_DigOut_C_7 AT %QX0.18744.0:BOOL;	(* Digital output value bit 7 MPNC020 02 module C *)
	MPNC_DigOut_C_8 AT %QX0.18748.0:BOOL;	(* Digital output value bit 8 MPNC020 02 module C *)
	MPNC_DigOut_C_9 AT %QX0.18752.0:BOOL;	(* Digital output value bit 9 MPNC020 02 module C *)
	MPNC_DigOut_C_10 AT %QX0.18756.0:BOOL;	(* Digital output value bit 10 MPNC020 02 module C *)
	MPNC_DigOut_C_11 AT %QX0.18760.0:BOOL;	(* Digital output value bit 11 MPNC020 02 module C *)
	MPNC_DigOut_C_12 AT %QX0.18764.0:BOOL;	(* Digital output value bit 12 MPNC020 02 module C *)
	MPNC_DigOut_C_13 AT %QX0.18768.0:BOOL;	(* Digital output value bit 13 MPNC020 02 module C *)
	MPNC_DigOut_C_14 AT %QX0.18772.0:BOOL;	(* Digital output value bit 14 MPNC020 02 module C *)
	MPNC_DigOut_C_15 AT %QX0.18776.0:BOOL;	(* Digital output value bit 15 MPNC020 02 module C *)
	MPNC_DigOut_C_16 AT %QX0.18780.0:BOOL;	(* Digital output value bit 16 MPNC020 02 module C *)
	MPNC_DigIn_A_1 AT %IX0.18848.0:BOOL;	(* Digital input value bit 1 MPNC020 01 module A *)
	MPNC_DigIn_A_2 AT %IX0.18852.0:BOOL;	(* Digital input value bit 2 MPNC020 01 module A *)
	MPNC_DigIn_A_3 AT %IX0.18856.0:BOOL;	(* Digital input value bit 3 MPNC020 01 module A *)
	MPNC_DigIn_A_4 AT %IX0.18860.0:BOOL;	(* Digital input value bit 4 MPNC020 01 module A *)
	MPNC_DigIn_A_5 AT %IX0.18864.0:BOOL;	(* Digital input value bit 5 MPNC020 01 module A *)
	MPNC_DigIn_A_6 AT %IX0.18868.0:BOOL;	(* Digital input value bit 6 MPNC020 01 module A *)
	MPNC_DigIn_A_7 AT %IX0.18872.0:BOOL;	(* Digital input value bit 7 MPNC020 01 module A *)
	MPNC_DigIn_A_8 AT %IX0.18876.0:BOOL;	(* Digital input value bit 8 MPNC020 01 module A *)
	MPNC_DigIn_A_9 AT %IX0.18880.0:BOOL;	(* Digital input value bit 9 MPNC020 01 module A *)
	MPNC_DigIn_A_10 AT %IX0.18884.0:BOOL;	(* Digital input value bit 10 MPNC020 01 module A *)
	MPNC_DigIn_A_11 AT %IX0.18888.0:BOOL;	(* Digital input value bit 11 MPNC020 01 module A *)
	MPNC_DigIn_A_12 AT %IX0.18892.0:BOOL;	(* Digital input value bit 12 MPNC020 01 module A *)
	MPNC_DigIn_A_13 AT %IX0.18896.0:BOOL;	(* Digital input value bit 13 MPNC020 01 module A *)
	MPNC_DigIn_A_14 AT %IX0.18900.0:BOOL;	(* Digital input value bit 14 MPNC020 01 module A *)
	MPNC_DigIn_A_15 AT %IX0.18904.0:BOOL;	(* Digital input value bit 15 MPNC020 01 module A *)
	MPNC_DigIn_A_16 AT %IX0.18908.0:BOOL;	(* Digital input value bit 16 MPNC020 01 module A *)
	MPNC_DigIn_B_1 AT %IX0.18912.0:BOOL;	(* Digital input value bit 1 MPNC020 01 module B *)
	MPNC_DigIn_B_2 AT %IX0.18916.0:BOOL;	(* Digital input value bit 2 MPNC020 01 module B *)
	MPNC_DigIn_B_3 AT %IX0.18920.0:BOOL;	(* Digital input value bit 3 MPNC020 01 module B *)
	MPNC_DigIn_B_4 AT %IX0.18924.0:BOOL;	(* Digital input value bit 4 MPNC020 01 module B *)
	MPNC_DigIn_B_5 AT %IX0.18928.0:BOOL;	(* Digital input value bit 5 MPNC020 01 module B *)
	MPNC_DigIn_B_6 AT %IX0.18932.0:BOOL;	(* Digital input value bit 6 MPNC020 01 module B *)
	MPNC_DigIn_B_7 AT %IX0.18936.0:BOOL;	(* Digital input value bit 7 MPNC020 01 module B *)
	MPNC_DigIn_B_8 AT %IX0.18940.0:BOOL;	(* Digital input value bit 8 MPNC020 01 module B *)
	MPNC_DigIn_B_9 AT %IX0.18944.0:BOOL;	(* Digital input value bit 9 MPNC020 01 module B *)
	MPNC_DigIn_B_10 AT %IX0.18948.0:BOOL;	(* Digital input value bit 10 MPNC020 01 module B *)
	MPNC_DigIn_B_11 AT %IX0.18952.0:BOOL;	(* Digital input value bit 11 MPNC020 01 module B *)
	MPNC_DigIn_B_12 AT %IX0.18956.0:BOOL;	(* Digital input value bit 12 MPNC020 01 module B *)
	MPNC_DigIn_B_13 AT %IX0.18960.0:BOOL;	(* Digital input value bit 13 MPNC020 01 module B *)
	MPNC_DigIn_B_14 AT %IX0.18964.0:BOOL;	(* Digital input value bit 14 MPNC020 01 module B *)
	MPNC_DigIn_B_15 AT %IX0.18968.0:BOOL;	(* Digital input value bit 15 MPNC020 01 module B *)
	MPNC_DigIn_B_16 AT %IX0.18972.0:BOOL;	(* Digital input value bit 16 MPNC020 01 module B *)
	MPNC_Reserved_1 AT %IW0.19104:UINT;
	MPNC_Reserved_2 AT %IW0.19108:UINT;
	MPNC_ColdJunctionT AT %IW0.19112:INT;	(* Cold junction temperature value *)
	MPNC_Reserved_3 AT %IW0.19116:UINT;
	MPNC_Reserved_4 AT %IW0.19120:UINT;
	MPNC_Reboot AT %QW0.19124:INT;	(* MPNC006 chain reboot *)
	MPNC_ModulesNumber AT %IW0.19128:UINT;	(* Number of modules *)
	MPNC_AnInConf_1 AT %QW0.19132:UINT;	(* Analog input 1 configuration MPNC006 *)
	MPNC_AnInConf_2 AT %QW0.19136:UINT;	(* Analog input 2 configuration MPNC006 *)
	MPNC_AnIn_1 AT %IW0.19140:INT;	(* Analog input 1 value MPNC006 *)
	MPNC_AnIn_2 AT %IW0.19144:INT;	(* Analog input 2 value MPNC006 *)
	MPNC_DigDir_1 AT %QX0.19148.0:BOOL;	(* Digital IO 1 configuration MPNC006 *)
	MPNC_DigDir_2 AT %QX0.19152.0:BOOL;	(* Digital IO 2 configuration MPNC006 *)
	MPNC_DigDir_3 AT %QX0.19156.0:BOOL;	(* Digital IO 3 configuration MPNC006 *)
	MPNC_DigDir_4 AT %QX0.19160.0:BOOL;	(* Digital IO 4 configuration MPNC006 *)
	MPNC_DigDir_5 AT %QX0.19164.0:BOOL;	(* Digital IO 5 configuration MPNC006 *)
	MPNC_DigDir_6 AT %QX0.19168.0:BOOL;	(* Digital IO 6 configuration MPNC006 *)
	MPNC_DigDir_7 AT %QX0.19172.0:BOOL;	(* Digital IO 7 configuration MPNC006 *)
	MPNC_DigDir_8 AT %QX0.19176.0:BOOL;	(* Digital IO 8 configuration MPNC006 *)
	MPNC_DigIn_1 AT %IX0.19180.0:BOOL;	(* Digital input 1 value MPNC006 *)
	MPNC_DigIn_2 AT %IX0.19184.0:BOOL;	(* Digital input 2 value MPNC006 *)
	MPNC_DigIn_3 AT %IX0.19188.0:BOOL;	(* Digital input 3 value MPNC006 *)
	MPNC_DigIn_4 AT %IX0.19192.0:BOOL;	(* Digital input 4 value MPNC006 *)
	MPNC_DigIn_5 AT %IX0.19196.0:BOOL;	(* Digital input 5 value MPNC006 *)
	MPNC_DigIn_6 AT %IX0.19200.0:BOOL;	(* Digital input 6 value MPNC006 *)
	MPNC_DigIn_7 AT %IX0.19204.0:BOOL;	(* Digital input 7 value MPNC006 *)
	MPNC_DigIn_8 AT %IX0.19208.0:BOOL;	(* Digital input 8 value MPNC006 *)
	MPNC_DigOut_1 AT %QX0.19212.0:BOOL;	(* Digital output 1 value MPNC006 *)
	MPNC_DigOut_2 AT %QX0.19216.0:BOOL;	(* Digital output 2 value MPNC006 *)
	MPNC_DigOut_3 AT %QX0.19220.0:BOOL;	(* Digital output 3 value MPNC006 *)
	MPNC_DigOut_4 AT %QX0.19224.0:BOOL;	(* Digital output 4 value MPNC006 *)
	MPNC_DigOut_5 AT %QX0.19228.0:BOOL;	(* Digital output 5 value MPNC006 *)
	MPNC_DigOut_6 AT %QX0.19232.0:BOOL;	(* Digital output 6 value MPNC006 *)
	MPNC_DigOut_7 AT %QX0.19236.0:BOOL;	(* Digital output 7 value MPNC006 *)
	MPNC_DigOut_8 AT %QX0.19240.0:BOOL;	(* Digital output 8 value MPNC006 *)
	MPNC_AnInFltr_1 AT %QW0.19244:UINT;	(* Analog input filter 1 MPNC006 *)
	MPNC_AnInFltr_2 AT %QW0.19248:UINT;	(* Analog input filter 2 MPNC006 *)
	MPNC_WatchDog AT %QW0.19252:UINT;	(* WatchDog Timer in Seconds *)
	MPNC_Reserved_6 AT %IW0.19272:UINT;
	MPNC_FirmwareVer AT %IW0.19340:UINT;	(* Firmware release MPNC006 *)
	MPNC_StatusWord AT %IW0.19344:UINT;	(* Status word MPNC006 *)
	RTU_StatusWord_1 AT %IW0.19348:UINT;
	RTU_BitMask_1 AT %ID0.19352:UDINT;
	RTU_HeartBeat_1 AT %ID0.19356:UDINT;
	RTU_temperature AT %IW0.19360:INT;
	RTU_humidity AT %IW0.19364:INT;
	RTU_CO2 AT %IW0.19368:INT;
	RTU_O3 AT %IW0.19372:INT;
	RTU_VOC AT %IW0.19376:INT;
	RTU_PM_1_0_C AT %IW0.19380:INT;
	RTU_PM_2_5_C AT %IW0.19384:INT;
	RTU_PM_4_0_C AT %IW0.19388:INT;
	RTU_PM_10_C AT %IW0.19392:INT;
	RTU_PM_1_0_N AT %IW0.19396:INT;
	RTU_PM_2_5_N AT %IW0.19400:INT;
	RTU_PM_4_0_N AT %IW0.19404:INT;
	RTU_PM_10_N AT %IW0.19408:INT;
	RTU_MPD AT %IW0.19412:INT;
	RTU_P AT %IW0.19416:INT;
	RTU_r16 AT %IW0.19420:INT;
	RTU_r17 AT %IW0.19424:INT;
	RTU_r18 AT %IW0.19428:INT;
	RTU_r19 AT %IW0.19432:INT;
	RTU_r20 AT %IW0.19436:INT;
	RTU_r21 AT %IW0.19440:INT;
	RTU_r22 AT %IW0.19444:INT;
	RTU_r23 AT %IW0.19448:INT;
	RTU_r24 AT %IW0.19452:INT;
	RTU_r25 AT %IW0.19456:INT;
	RTU_r26 AT %IW0.19460:INT;
	RTU_r27 AT %IW0.19464:INT;
	RTU_r28 AT %IW0.19468:INT;
	RTU_r29 AT %IW0.19472:INT;
	RTU_r30 AT %IW0.19476:INT;
	RTU_r31 AT %IW0.19480:INT;
	RTU_r32 AT %IW0.19484:INT;
	RTU_StatusWord_2 AT %IW0.19488:UINT;
	RTU_BitMask_2 AT %ID0.19492:UDINT;
	RTU_HeartBeat_2 AT %ID0.19496:UDINT;
	RTU_temperature_bis AT %IW0.19500:INT;
	RTU_humidity_bis AT %IW0.19504:INT;
	RTU_StatusWord_3 AT %IW0.19508:UINT;
	RTU_BitMask_3 AT %ID0.19512:UDINT;
	RTU_HeartBeat_3 AT %ID0.19516:UDINT;
	RTU_temperature_ext AT %IW0.19520:INT;
	RTU_humidity_ext AT %IW0.19524:INT;
	PLC_FWrevision AT %IW0.19528:UINT;	(* Firmware version *)
	PLC_HWconfig AT %IW0.19532:UINT;	(* Hardware configuration *)
	PLC_DigDir_1 AT %QX0.19536.0:BOOL;	(* Digital 1 direction (input = 0 output = 1) *)
	PLC_DigDir_2 AT %QX0.19540.0:BOOL;	(* Digital 2 direction (input = 0 output = 1) *)
	PLC_DigDir_3 AT %QX0.19544.0:BOOL;	(* Digital 3 direction (input = 0 output = 1) *)
	PLC_DigDir_4 AT %QX0.19548.0:BOOL;	(* Digital 4 direction (input = 0 output = 1) *)
	PLC_DigDir_5 AT %QX0.19552.0:BOOL;	(* Digital 5 direction (input = 0 output = 1) *)
	PLC_DigDir_6 AT %QX0.19556.0:BOOL;	(* Digital 6 direction (input = 0 output = 1) *)
	PLC_DigDir_7 AT %QX0.19560.0:BOOL;	(* Digital 7 direction (input = 0 output = 1) *)
	PLC_DigDir_8 AT %QX0.19564.0:BOOL;	(* Digital 8 direction (input = 0 output = 1) *)
	PLC_AnInConf_1 AT %QW0.19568:UINT;	(* Analog input 1 configuration *)
	PLC_AnInConf_2 AT %QW0.19572:UINT;	(* Analog input 2 configuration *)
	PLC_AnOutConf_1 AT %QW0.19576:UINT;	(* Analog output 1 configuration *)
	PLC_AnOutConf_2 AT %QW0.19580:UINT;	(* Analog output 2 configuration *)
	PLC_AnInConf_3 AT %QW0.19584:UINT;	(* Analog input 3 configuration *)
	PLC_Reserved_1 AT %QW0.19588:UINT;	(* Reserved *)
	PLC_DigIn_1 AT %IX0.19592.0:BOOL;	(* Digital input 1 value *)
	PLC_DigIn_2 AT %IX0.19596.0:BOOL;	(* Digital input 2 value *)
	PLC_DigIn_3 AT %IX0.19600.0:BOOL;	(* Digital input 3 value *)
	PLC_DigIn_4 AT %IX0.19604.0:BOOL;	(* Digital input 4 value *)
	PLC_DigIn_5 AT %IX0.19608.0:BOOL;	(* Digital input 5 value *)
	PLC_DigIn_6 AT %IX0.19612.0:BOOL;	(* Digital input 6 value *)
	PLC_DigIn_7 AT %IX0.19616.0:BOOL;	(* Digital input 7 value *)
	PLC_DigIn_8 AT %IX0.19620.0:BOOL;	(* Digital input 8 value *)
	PLC_DigIn_9 AT %IX0.19624.0:BOOL;	(* Digital input 9 value *)
	PLC_DigIn_10 AT %IX0.19628.0:BOOL;	(* Digital input 10 value *)
	PLC_DigIn_11 AT %IX0.19632.0:BOOL;	(* Digital input 11 value *)
	PLC_DigIn_12 AT %IX0.19636.0:BOOL;	(* Digital input 12 value *)
	PLC_AnIn_1 AT %IW0.19640:INT;	(* Analog input 1 value *)
	PLC_AnIn_2 AT %IW0.19644:INT;	(* Analog input 2 value *)
	PLC_AnIn_3 AT %IW0.19648:INT;	(* Analog input 3 value *)
	PLC_Reserved_2 AT %IW0.19652:INT;	(* Reserved *)
	PLC_Reserved_3 AT %IW0.19656:INT;	(* Reserved *)
	PLC_Tamb AT %IW0.19660:INT;	(* Cold junction compensation value *)
	PLC_Encoder AT %ID0.19664:DINT;	(* Encoder reading value *)
	PLC_Capture AT %ID0.19668:UDINT;	(* Time between 2 input edges *)
	PLC_DigOut_1 AT %QX0.19672.0:BOOL;	(* Digital output 1 value *)
	PLC_DigOut_2 AT %QX0.19676.0:BOOL;	(* Digital output 2 value *)
	PLC_DigOut_3 AT %QX0.19680.0:BOOL;	(* Digital output 3 value *)
	PLC_DigOut_4 AT %QX0.19684.0:BOOL;	(* Digital output 4 value *)
	PLC_DigOut_5 AT %QX0.19688.0:BOOL;	(* Digital output 5 value *)
	PLC_DigOut_6 AT %QX0.19692.0:BOOL;	(* Digital output 6 value *)
	PLC_DigOut_7 AT %QX0.19696.0:BOOL;	(* Digital output 7 value *)
	PLC_DigOut_8 AT %QX0.19700.0:BOOL;	(* Digital output 8 value *)
	PLC_AnOut_1 AT %QW0.19704:INT;	(* Analog output 1 value *)
	PLC_AnOut_2 AT %QW0.19708:INT;	(* Analog output 2 value *)
	PLC_Reserved_4 AT %QW0.19712:INT;	(* Reserved *)
	PLC_Reserved_5 AT %QW0.19716:INT;	(* Reserved *)
	PLC_EncoderStart AT %QW0.19720:UINT;	(* Encoder - counter enable *)
	PLC_EncoderReset AT %QW0.19724:UINT;	(* Encoder reset *)
	PLC_Heartbeat AT %IW0.19728:UINT;	(* In - Out board function check *)
	PLC_StatusReg AT %IW0.19732:UINT;	(* In - Out board status *)
	PLC_AnIn1Filter AT %QW0.19736:UINT;	(* Analog input 1 filter *)
	PLC_AnIn2Filter AT %QW0.19740:UINT;	(* Analog input 2 filter *)
	PLC_AnIn3Filter AT %QW0.19744:UINT;	(* Analog input 3 filter *)
	PLC_Reserved_6 AT %QW0.19748:UINT;	(* Reserved *)
	PLC_Reserved_7 AT %QW0.19752:UINT;	(* Reserved *)
	SysActivePower_0 AT %ID0.19756:REAL;	(* 0x0A 0x1026 Potenza Attiva 0 in W (PRINCIPALE) *)
	SysActivePower_1 AT %ID0.19760:REAL;	(* 0x0B 0x1026 Potenza Attiva 0 in W (PRINCIPALE) *)
	SysActivePower_2 AT %ID0.19764:REAL;	(* 0x0C 0x1026 Potenza Attiva 0 in W (ESTERNI) *)
	SysActivePower_3 AT %ID0.19768:REAL;	(* 0x0D 0x1026 Potenza Attiva 0 in W (PIANO SOPRA) *)
	SysActivePower_4 AT %ID0.19772:REAL;	(* 0x0E 0x1026 Potenza Attiva 0 in W (PIANO TERRA) *)
	SysActivePower_5 AT %ID0.19776:REAL;	(* 0x0F 0x1026 Potenza Attiva 0 in W (PIANO SOTTO) *)
	SysActivePower_6 AT %ID0.19780:REAL;	(* 0x10 0x1026 Potenza Attiva 0 in W (AUTO ELETTRICA) *)
	SysActivePower_7 AT %ID0.19784:REAL;	(* 0x11 0x1026 Potenza Attiva 0 in W (DEUMIDIFICATORE) *)
	SysActivePower_8 AT %ID0.19788:REAL;	(* 0x12 0x1026 Potenza Attiva 0 in W (LAVANDERIA) *)
	SysActivePower_9 AT %ID0.19792:REAL;	(* 0x13 0x1026 Potenza Attiva 0 in W (UPS) *)
	SysActivePower_10 AT %ID0.19796:REAL;	(* 0x14 0x1026 Potenza Attiva 0 in W (Puffer) *)
	SysActivePower_11 AT %QD0.19800:REAL;	(* 0x15 0x1026 Potenza Attiva 0 in W (Caldaia) *)
	SysApparentPower_0 AT %ID0.19804:REAL;	(* 0x0A 0x102E Potenza Apparente 0 in VA (UPS) *)
	SysApparentPower_1 AT %ID0.19808:REAL;	(* 0x0B 0x102E Potenza Apparente 0 in VA (UPS) *)
	SysApparentPower_2 AT %ID0.19812:REAL;	(* 0x0C 0x102E Potenza Apparente 0 in VA (UPS) *)
	SysApparentPower_3 AT %ID0.19816:REAL;	(* 0x0D 0x102E Potenza Apparente 0 in VA (UPS) *)
	SysApparentPower_4 AT %ID0.19820:REAL;	(* 0x0E 0x102E Potenza Apparente 0 in VA (UPS) *)
	SysApparentPower_5 AT %ID0.19824:REAL;	(* 0x0F 0x102E Potenza Apparente 0 in VA (UPS) *)
	SysApparentPower_6 AT %ID0.19828:REAL;	(* 0x10 0x102E Potenza Apparente 0 in VA (UPS) *)
	SysApparentPower_7 AT %ID0.19832:REAL;	(* 0x11 0x102E Potenza Apparente 0 in VA (UPS) *)
	SysApparentPower_8 AT %ID0.19836:REAL;	(* 0x12 0x102E Potenza Apparente 0 in VA (UPS) *)
	SysApparentPower_9 AT %ID0.19840:REAL;	(* 0x13 0x102E Potenza Apparente 0 in VA (UPS) *)
	SysApparentPower_10 AT %ID0.19844:REAL;	(* 0x14 0x102E Potenza Apparente 0 in VA (UPS) *)
	SysApparentPower_11 AT %ID0.19848:REAL;	(* 0x15 0x102E Potenza Apparente 0 in VA (UPS) *)
	SysExpActiveEnergy_0 AT %ID0.19852:REAL;	(* 0x0A 0x110E Energia Attiva Esportata 0 in Wh (PRINCIPALE) *)
	SysExpActiveEnergy_1 AT %ID0.19856:REAL;	(* 0x0B 0x110E Energia Attiva Esportata 0 in Wh (PRINCIPALE) *)
	SysImpActiveEnergy_0 AT %ID0.19860:REAL;	(* 0x0A 0x1106 Energia Attiva Importata 0 in Wh (PRINCIPALE) *)
	SysImpActiveEnergy_1 AT %ID0.19864:REAL;	(* 0x0B 0x1106 Energia Attiva Importata 0 in Wh (PRINCIPALE) *)
	SysImpActiveEnergy_2 AT %ID0.19868:REAL;	(* 0x0C 0x1106 Energia Attiva Importata 0 in Wh (UPS) *)
	SysImpActiveEnergy_3 AT %ID0.19872:REAL;	(* 0x0D 0x1106 Energia Attiva Importata 0 in Wh (UPS) *)
	SysImpActiveEnergy_4 AT %ID0.19876:REAL;	(* 0x0E 0x1106 Energia Attiva Importata 0 in Wh (UPS) *)
	SysImpActiveEnergy_5 AT %ID0.19880:REAL;	(* 0x0F 0x1106 Energia Attiva Importata 0 in Wh (UPS) *)
	SysImpActiveEnergy_6 AT %ID0.19884:REAL;	(* 0x10 0x1106 Energia Attiva Importata 0 in Wh (UPS) *)
	SysImpActiveEnergy_7 AT %ID0.19888:REAL;	(* 0x11 0x1106 Energia Attiva Importata 0 in Wh (UPS) *)
	SysImpActiveEnergy_8 AT %ID0.19892:REAL;	(* 0x12 0x1106 Energia Attiva Importata 0 in Wh (UPS) *)
	SysImpActiveEnergy_9 AT %ID0.19896:REAL;	(* 0x13 0x1106 Energia Attiva Importata 0 in Wh (UPS) *)
	SysImpActiveEnergy_10 AT %ID0.19900:REAL;	(* 0x14 0x1106 Energia Attiva Importata 0 in Wh (UPS) *)
	SysImpActiveEnergy_11 AT %ID0.19904:REAL;	(* 0x15 0x1106 Energia Attiva Importata 0 in Wh (UPS) *)
	SysPowerFactor_0 AT %ID0.19908:REAL;	(* 0x0A 0x101E Fattore di Potenza 0 (PRINCIPALE) *)
	SysPowerFactor_1 AT %ID0.19912:REAL;	(* 0x0B 0x101E Fattore di Potenza 0 (PRINCIPALE) *)
	SysReactivePower_0 AT %ID0.19916:REAL;	(* 0x0A 0x1036 Potenza Reattiva 0 in var *)
	Frequency_0 AT %ID0.19920:REAL;	(* 0x0A 0x1038 Frequenza in Hz *)
	SysReactivePower_1 AT %ID0.19924:REAL;	(* 0x0B 0x1036 Potenza Reattiva 0 in var *)
	SysReactivePower_2 AT %ID0.19932:REAL;	(* 0x0C 0x1036 Potenza Reattiva 0 in var *)
	SysReactivePower_3 AT %ID0.19936:REAL;	(* 0x0D 0x1036 Potenza Reattiva 0 in var *)
	SysReactivePower_4 AT %ID0.19940:REAL;	(* 0x0E 0x1036 Potenza Reattiva 0 in var *)
	SysReactivePower_5 AT %ID0.19944:REAL;	(* 0x0F 0x1036 Potenza Reattiva 0 in var *)
	SysReactivePower_6 AT %ID0.19948:REAL;	(* 0x10 0x1036 Potenza Reattiva 0 in var *)
	SysReactivePower_7 AT %ID0.19952:REAL;	(* 0x11 0x1036 Potenza Reattiva 0 in var *)
	SysReactivePower_8 AT %ID0.19956:REAL;	(* 0x12 0x1036 Potenza Reattiva 0 in var *)
	SysReactivePower_9 AT %ID0.19960:REAL;	(* 0x13 0x1036 Potenza Reattiva 0 in var *)
	SysReactivePower_10 AT %ID0.19964:REAL;	(* 0x14 0x1036 Potenza Reattiva 0 in var *)
	SysReactivePower_11 AT %ID0.19968:REAL;	(* 0x15 0x1036 Potenza Reattiva 0 in var *)
	SystemCurrent_0 AT %ID0.19972:REAL;	(* 0x0A 0x1016 Corrente in A *)
	SystemVoltage_0 AT %ID0.19980:REAL;	(* 0x0A 0x100C Tensione in V (PRINCIPALE) *)
	RTU0_TYPE_PORT AT %ID0.20000:UDINT;
	RTU0_BAUDRATE AT %ID0.20004:UDINT;
	RTU0_STATUS AT %ID0.20008:UDINT;
	RTU0_READS AT %ID0.20012:UDINT;
	RTU0_WRITES AT %ID0.20016:UDINT;
	RTU0_TIMEOUTS AT %ID0.20020:UDINT;
	RTU0_COMM_ERRORS AT %ID0.20024:UDINT;
	RTU0_LAST_ERROR AT %ID0.20028:UDINT;
	RTU0_WRITE_QUEUE AT %ID0.20032:UDINT;
	RTU0_BUS_LOAD AT %ID0.20036:UDINT;
	RTU3_TYPE_PORT AT %ID0.20080:UDINT;
	RTU3_BAUDRATE AT %ID0.20084:UDINT;
	RTU3_STATUS AT %ID0.20088:UDINT;
	RTU3_READS AT %ID0.20092:UDINT;
	RTU3_WRITES AT %ID0.20096:UDINT;
	RTU3_TIMEOUTS AT %ID0.20100:UDINT;
	RTU3_COMM_ERRORS AT %ID0.20104:UDINT;
	RTU3_LAST_ERROR AT %ID0.20108:UDINT;
	RTU3_WRITE_QUEUE AT %ID0.20112:UDINT;
	RTU3_BUS_LOAD AT %ID0.20116:UDINT;
	TCPS_TYPE_PORT AT %ID0.20200:UDINT;
	TCPS_IP_ADDRESS AT %ID0.20204:UDINT;
	TCPS_STATUS AT %ID0.20208:UDINT;
	TCPS_READS AT %ID0.20212:UDINT;
	TCPS_WRITES AT %ID0.20216:UDINT;
	TCPS_TIMEOUTS AT %ID0.20220:UDINT;
	TCPS_COMM_ERRORS AT %ID0.20224:UDINT;
	TCPS_LAST_ERROR AT %ID0.20228:UDINT;
	TCPS_WRITE_QUEUE AT %ID0.20232:UDINT;
	TCPS_BUS_LOAD AT %ID0.20236:UDINT;
	TCP0_TYPE_PORT AT %ID0.20240:UDINT;
	TCP0_IP_ADDRESS AT %ID0.20244:UDINT;
	TCP0_STATUS AT %ID0.20248:UDINT;
	TCP0_READS AT %ID0.20252:UDINT;
	TCP0_WRITES AT %ID0.20256:UDINT;
	TCP0_TIMEOUTS AT %ID0.20260:UDINT;
	TCP0_COMM_ERRORS AT %ID0.20264:UDINT;
	TCP0_LAST_ERROR AT %ID0.20268:UDINT;
	TCP0_WRITE_QUEUE AT %ID0.20272:UDINT;
	TCP0_BUS_LOAD AT %ID0.20276:UDINT;
	TCP1_TYPE_PORT AT %ID0.20280:UDINT;
	TCP1_IP_ADDRESS AT %ID0.20284:UDINT;
	TCP1_STATUS AT %ID0.20288:UDINT;
	TCP1_READS AT %ID0.20292:UDINT;
	TCP1_WRITES AT %ID0.20296:UDINT;
	TCP1_TIMEOUTS AT %ID0.20300:UDINT;
	TCP1_COMM_ERRORS AT %ID0.20304:UDINT;
	TCP1_LAST_ERROR AT %ID0.20308:UDINT;
	TCP1_WRITE_QUEUE AT %ID0.20312:UDINT;
	TCP1_BUS_LOAD AT %ID0.20316:UDINT;
	TCP2_TYPE_PORT AT %ID0.20320:UDINT;
	TCP2_IP_ADDRESS AT %ID0.20324:UDINT;
	TCP2_STATUS AT %ID0.20328:UDINT;
	TCP2_READS AT %ID0.20332:UDINT;
	TCP2_WRITES AT %ID0.20336:UDINT;
	TCP2_TIMEOUTS AT %ID0.20340:UDINT;
	TCP2_COMM_ERRORS AT %ID0.20344:UDINT;
	TCP2_LAST_ERROR AT %ID0.20348:UDINT;
	TCP2_WRITE_QUEUE AT %ID0.20352:UDINT;
	TCP2_BUS_LOAD AT %ID0.20356:UDINT;
	TCP3_TYPE_PORT AT %ID0.20360:UDINT;
	TCP3_IP_ADDRESS AT %ID0.20364:UDINT;
	TCP3_STATUS AT %ID0.20368:UDINT;
	TCP3_READS AT %ID0.20372:UDINT;
	TCP3_WRITES AT %ID0.20376:UDINT;
	TCP3_TIMEOUTS AT %ID0.20380:UDINT;
	TCP3_COMM_ERRORS AT %ID0.20384:UDINT;
	TCP3_LAST_ERROR AT %ID0.20388:UDINT;
	TCP3_WRITE_QUEUE AT %ID0.20392:UDINT;
	TCP3_BUS_LOAD AT %ID0.20396:UDINT;
	TCP4_TYPE_PORT AT %ID0.20400:UDINT;
	TCP4_IP_ADDRESS AT %ID0.20404:UDINT;
	TCP4_STATUS AT %ID0.20408:UDINT;
	TCP4_READS AT %ID0.20412:UDINT;
	TCP4_WRITES AT %ID0.20416:UDINT;
	TCP4_TIMEOUTS AT %ID0.20420:UDINT;
	TCP4_COMM_ERRORS AT %ID0.20424:UDINT;
	TCP4_LAST_ERROR AT %ID0.20428:UDINT;
	TCP4_WRITE_QUEUE AT %ID0.20432:UDINT;
	TCP4_BUS_LOAD AT %ID0.20436:UDINT;
	TCP5_TYPE_PORT AT %ID0.20440:UDINT;
	TCP5_IP_ADDRESS AT %ID0.20444:UDINT;
	TCP5_STATUS AT %ID0.20448:UDINT;
	TCP5_READS AT %ID0.20452:UDINT;
	TCP5_WRITES AT %ID0.20456:UDINT;
	TCP5_TIMEOUTS AT %ID0.20460:UDINT;
	TCP5_COMM_ERRORS AT %ID0.20464:UDINT;
	TCP5_LAST_ERROR AT %ID0.20468:UDINT;
	TCP5_WRITE_QUEUE AT %ID0.20472:UDINT;
	TCP5_BUS_LOAD AT %ID0.20476:UDINT;
	TCP6_TYPE_PORT AT %ID0.20480:UDINT;
	TCP6_IP_ADDRESS AT %ID0.20484:UDINT;
	TCP6_STATUS AT %ID0.20488:UDINT;
	TCP6_READS AT %ID0.20492:UDINT;
	TCP6_WRITES AT %ID0.20496:UDINT;
	TCP6_TIMEOUTS AT %ID0.20500:UDINT;
	TCP6_COMM_ERRORS AT %ID0.20504:UDINT;
	TCP6_LAST_ERROR AT %ID0.20508:UDINT;
	TCP6_WRITE_QUEUE AT %ID0.20512:UDINT;
	TCP6_BUS_LOAD AT %ID0.20516:UDINT;
	TCP7_TYPE_PORT AT %ID0.20520:UDINT;
	TCP7_IP_ADDRESS AT %ID0.20524:UDINT;
	TCP7_STATUS AT %ID0.20528:UDINT;
	TCP7_READS AT %ID0.20532:UDINT;
	TCP7_WRITES AT %ID0.20536:UDINT;
	TCP7_TIMEOUTS AT %ID0.20540:UDINT;
	TCP7_COMM_ERRORS AT %ID0.20544:UDINT;
	TCP7_LAST_ERROR AT %ID0.20548:UDINT;
	TCP7_WRITE_QUEUE AT %ID0.20552:UDINT;
	TCP7_BUS_LOAD AT %ID0.20556:UDINT;
	NODE_01_DEV_NODE AT %QD0.20688:UDINT;
	NODE_01_STATUS AT %QD0.20692:UDINT;
	NODE_02_DEV_NODE AT %QD0.20696:UDINT;
	NODE_02_STATUS AT %QD0.20700:UDINT;
	NODE_03_DEV_NODE AT %QD0.20704:UDINT;
	NODE_03_STATUS AT %QD0.20708:UDINT;
	NODE_04_DEV_NODE AT %QD0.20712:UDINT;
	NODE_04_STATUS AT %QD0.20716:UDINT;
	NODE_05_DEV_NODE AT %QD0.20720:UDINT;
	NODE_05_STATUS AT %QD0.20724:UDINT;
	NODE_06_DEV_NODE AT %QD0.20728:UDINT;
	NODE_06_STATUS AT %QD0.20732:UDINT;
	NODE_07_DEV_NODE AT %QD0.20736:UDINT;
	NODE_07_STATUS AT %QD0.20740:UDINT;
	NODE_08_DEV_NODE AT %QD0.20744:UDINT;
	NODE_08_STATUS AT %QD0.20748:UDINT;
	NODE_09_DEV_NODE AT %QD0.20752:UDINT;
	NODE_09_STATUS AT %QD0.20756:UDINT;
	NODE_10_DEV_NODE AT %QD0.20760:UDINT;
	NODE_10_STATUS AT %QD0.20764:UDINT;
	NODE_11_DEV_NODE AT %QD0.20768:UDINT;
	NODE_11_STATUS AT %QD0.20772:UDINT;
	NODE_12_DEV_NODE AT %QD0.20776:UDINT;
	NODE_12_STATUS AT %QD0.20780:UDINT;
	NODE_13_DEV_NODE AT %QD0.20784:UDINT;
	NODE_13_STATUS AT %QD0.20788:UDINT;
	NODE_14_DEV_NODE AT %QD0.20792:UDINT;
	NODE_14_STATUS AT %QD0.20796:UDINT;
	NODE_15_DEV_NODE AT %QD0.20800:UDINT;
	NODE_15_STATUS AT %QD0.20804:UDINT;
	NODE_16_DEV_NODE AT %QD0.20808:UDINT;
	NODE_16_STATUS AT %QD0.20812:UDINT;
	NODE_17_DEV_NODE AT %QD0.20816:UDINT;
	NODE_17_STATUS AT %QD0.20820:UDINT;
	NODE_18_DEV_NODE AT %QD0.20824:UDINT;
	NODE_18_STATUS AT %QD0.20828:UDINT;
	NODE_19_DEV_NODE AT %QD0.20832:UDINT;
	NODE_19_STATUS AT %QD0.20836:UDINT;
	NODE_20_DEV_NODE AT %QD0.20840:UDINT;
	NODE_20_STATUS AT %QD0.20844:UDINT;
	NODE_21_DEV_NODE AT %QD0.20848:UDINT;
	NODE_21_STATUS AT %QD0.20852:UDINT;
	NODE_22_DEV_NODE AT %QD0.20856:UDINT;
	NODE_22_STATUS AT %QD0.20860:UDINT;
	NODE_23_DEV_NODE AT %QD0.20864:UDINT;
	NODE_23_STATUS AT %QD0.20868:UDINT;
	NODE_24_DEV_NODE AT %QD0.20872:UDINT;
	NODE_24_STATUS AT %QD0.20876:UDINT;
	NODE_25_DEV_NODE AT %QD0.20880:UDINT;
	NODE_25_STATUS AT %QD0.20884:UDINT;
	NODE_26_DEV_NODE AT %QD0.20888:UDINT;
	NODE_26_STATUS AT %QD0.20892:UDINT;
	NODE_27_DEV_NODE AT %QD0.20896:UDINT;
	NODE_27_STATUS AT %QD0.20900:UDINT;
	NODE_28_DEV_NODE AT %QD0.20904:UDINT;
	NODE_28_STATUS AT %QD0.20908:UDINT;
	NODE_29_DEV_NODE AT %QD0.20912:UDINT;
	NODE_29_STATUS AT %QD0.20916:UDINT;
	NODE_30_DEV_NODE AT %QD0.20920:UDINT;
	NODE_30_STATUS AT %QD0.20924:UDINT;
	NODE_31_DEV_NODE AT %QD0.20928:UDINT;
	NODE_31_STATUS AT %QD0.20932:UDINT;
	NODE_32_DEV_NODE AT %QD0.20936:UDINT;
	NODE_32_STATUS AT %QD0.20940:UDINT;
	NODE_33_DEV_NODE AT %QD0.20944:UDINT;
	NODE_33_STATUS AT %QD0.20948:UDINT;
	NODE_34_DEV_NODE AT %QD0.20952:UDINT;
	NODE_34_STATUS AT %QD0.20956:UDINT;
	NODE_35_DEV_NODE AT %QD0.20960:UDINT;
	NODE_35_STATUS AT %QD0.20964:UDINT;
	NODE_36_DEV_NODE AT %QD0.20968:UDINT;
	NODE_36_STATUS AT %QD0.20972:UDINT;
	NODE_37_DEV_NODE AT %QD0.20976:UDINT;
	NODE_37_STATUS AT %QD0.20980:UDINT;
	NODE_38_DEV_NODE AT %QD0.20984:UDINT;
	NODE_38_STATUS AT %QD0.20988:UDINT;
	NODE_39_DEV_NODE AT %QD0.20992:UDINT;
	NODE_39_STATUS AT %QD0.20996:UDINT;
	NODE_40_DEV_NODE AT %QD0.21000:UDINT;
	NODE_40_STATUS AT %QD0.21004:UDINT;
	NODE_41_DEV_NODE AT %QD0.21008:UDINT;
	NODE_41_STATUS AT %QD0.21012:UDINT;
	NODE_42_DEV_NODE AT %QD0.21016:UDINT;
	NODE_42_STATUS AT %QD0.21020:UDINT;
	NODE_43_DEV_NODE AT %QD0.21024:UDINT;
	NODE_43_STATUS AT %QD0.21028:UDINT;
	NODE_44_DEV_NODE AT %QD0.21032:UDINT;
	NODE_44_STATUS AT %QD0.21036:UDINT;
	NODE_45_DEV_NODE AT %QD0.21040:UDINT;
	NODE_45_STATUS AT %QD0.21044:UDINT;
	PLC_time AT %ID0.21560:REAL;	(* Seconds since boot (reset each 24h) *)
	PLC_timeMin AT %ID0.21564:REAL;	(* 10 seconds window start *)
	PLC_timeMax AT %ID0.21568:REAL;	(* 10 seconds window stop *)
	PLC_timeWin AT %QD0.21572:REAL;	(* Graph display window *)
	PLC_Version AT %IW0.21576:UINT;	(* Run Time version *)
	PLC_EngineStatus AT %IW0.21580:UINT;	(* PLC status *)
	PLC_ResetValues AT %QX0.21584.0:BOOL;	(* Diagnostic variables reset *)
	PLC_buzzerOn AT %QX0.21588.0:BOOL;	(* Buzzer sound (enable = 1 disable = 0) *)
	PLC_PLC_Version AT %QW0.21592:UINT;	(* PLC application version *)
	PLC_HMI_Version AT %QW0.21596:UINT;	(* HMI application version *)
	PLC_Year AT %IW0.21640:UINT;	(* Currently year *)
	PLC_Month AT %IW0.21644:UINT;	(* Currently month *)
	PLC_Day AT %IW0.21648:UINT;	(* Currently day *)
	PLC_Hours AT %IW0.21652:UINT;	(* Currently hour *)
	PLC_Minutes AT %IW0.21656:UINT;	(* Currently minutes *)
	PLC_Seconds AT %IW0.21660:UINT;	(* Currently seconds *)
	PLC_UPTIME_s AT %ID0.21664:UDINT;	(* Uptime in seconds (wraps in 136 years) *)
	PLC_UPTIME_cs AT %ID0.21668:UDINT;	(* Uptime in centiseconds = 10 ms (wraps in 497 days) *)
	PLC_WATCHDOGEN AT %QX0.21672.0:BOOL;	(* Enable Watchdog *)
	PLC_WATCHDOG_ms AT %QD0.21676:UDINT;	(* Reset Watchdog timer *)
	PLC_PRODUCT_ID AT %ID0.21680:UDINT;	(* TP/TPAC/TPLC Product ID (Hex) *)
	PLC_SERIAL_NUMBER AT %ID0.21684:UDINT;	(* TP/TPAC/TPLC Serial Number *)
	PLC_HMI_PAGE AT %QD0.21688:DINT;	(* HMI Page (page100=0x00000100) *)
	PLC_BEEP_VOLUME AT %QB0.21740:BYTE;	(* Beep volume (when buzzerOn) *)
	PLC_TOUCH_VOLUME AT %QB0.21744:BYTE;	(* Touch volume *)
	PLC_ALARM_VOLUME AT %QB0.21748:BYTE;	(* Alarm volume (when alarm) *)
	PLC_BUZZER AT %QD0.21752:UDINT;	(* Enable dynamic buzzer sound (0x44332211 up=0x11(%) on=0x22(cs) off=0x33(cs) rep=0x44(times)) *)
	PLC_FastIO_Ena AT %QD0.21756:UDINT;	(* Not available *)
	PLC_FastIO_Dir AT %QD0.21760:UDINT;	(* Not available *)
	PLC_FastIO_1 AT %QX0.21764.0:BOOL;	(* Not available *)
	PLC_FastIO_2 AT %QX0.21768.0:BOOL;	(* Not available *)
	PLC_FastIO_3 AT %QX0.21772.0:BOOL;	(* Not available *)
	PLC_FastIO_4 AT %QX0.21776.0:BOOL;	(* Not available *)
	PLC_FastIO_5 AT %QX0.21780.0:BOOL;	(* Not available *)
	PLC_FastIO_6 AT %QX0.21784.0:BOOL;	(* Not available *)
	PLC_FastIO_7 AT %QX0.21788.0:BOOL;	(* Not available *)
	PLC_FastIO_8 AT %QX0.21792.0:BOOL;	(* Not available *)
END_VAR
